ABB RAPID module: P105.mod

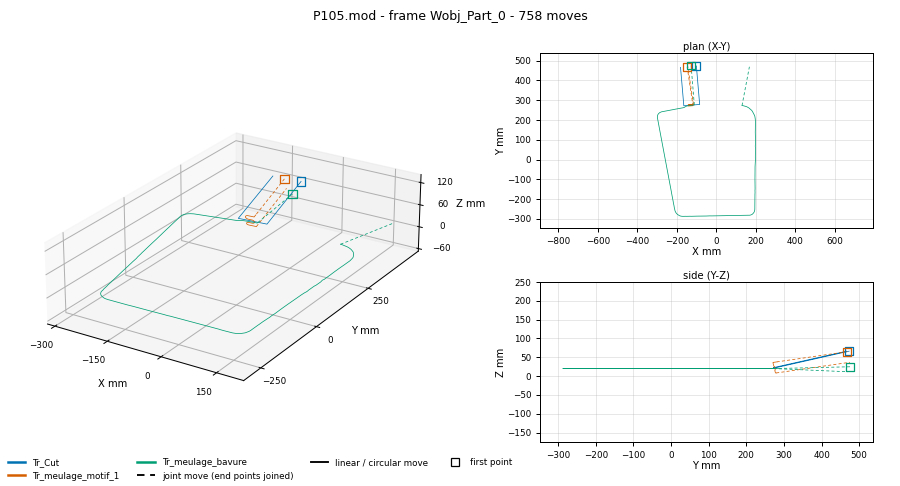
[picture p0: tool path of P105.mod in frame Wobj_Part_0, 758 of 766 moves have a stored position in this frame; points joined in program order, loops and branches not executed]
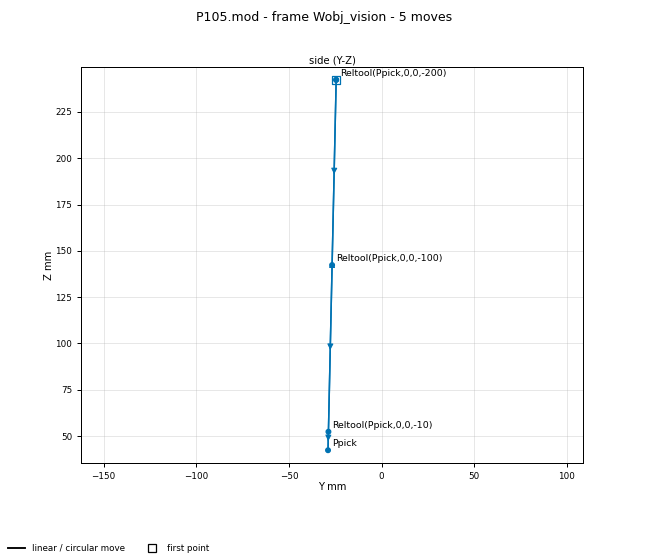
[picture p1: tool path of P105.mod in frame Wobj_vision, 5 of 766 moves have a stored position in this frame; points joined in program order, loops and branches not executed]
MODULE P105
	LOCAL CONST Speeddata vitesse_Tronconnage :=[10, 500, 0, 0];
	LOCAL CONST Robtarget Coupe_0 :=[[-129.483703125,274.966,22.39716015625],[0.465088414664095,0.570480739623642,-0.417793879465057,-0.532628169124803],[0,0,0,0],[8.999999E+09,8.999999E+09,8.999999E+09,8.999999E+09,8.999999E+09,8.999999E+09]];
	LOCAL CONST Robtarget Tr_meulage_motif_1_App1 :=[[-147.710429474566,468.187926503189,64.8611227493864],[0.0489177638432012,-0.0564309964361688,0.753506704297272,-0.653184691799237],[0,0,0,0],[8.999999E+09,8.999999E+09,8.999999E+09,8.999999E+09,8.999999E+09,8.999999E+09]];
	LOCAL CONST Robtarget Tr_meulage_motif_1_App2 :=[[-119.696933583103,282.208871325159,37.8975346530943],[0.0489177638432012,-0.0564309964361688,0.753506704297272,-0.653184691799237],[0,0,0,0],[8.999999E+09,8.999999E+09,8.999999E+09,8.999999E+09,8.999999E+09,8.999999E+09]];
	LOCAL CONST Robtarget Tr_meulage_motif_1_P0 :=[[-118.2225390625,272.4205,36.4783984375],[0.0489177638432012,-0.0564309964361688,0.753506704297272,-0.653184691799237],[0,0,0,0],[8.999999E+09,8.999999E+09,8.999999E+09,8.999999E+09,8.999999E+09,8.999999E+09]];
	LOCAL CONST Robtarget Tr_meulage_motif_1_P1 :=[[-119.2195859375,272.3438125,36.4796796875],[0.0489177638432012,-0.0564309964361688,0.753506704297272,-0.653184691799237],[0,0,0,0],[8.999999E+09,8.999999E+09,8.999999E+09,8.999999E+09,8.999999E+09,8.999999E+09]];
	LOCAL CONST Robtarget Tr_meulage_motif_1_P2 :=[[-120.216640625,272.267125,36.48095703125],[0.0489177638432012,-0.0564309964361688,0.753506704297272,-0.653184691799237],[0,0,0,0],[8.999999E+09,8.999999E+09,8.999999E+09,8.999999E+09,8.999999E+09,8.999999E+09]];
	LOCAL CONST Robtarget Tr_meulage_motif_1_P3 :=[[-121.2136953125,272.19040625,36.482234375],[0.0489177638432012,-0.0564309964361688,0.753506704297272,-0.653184691799237],[0,0,0,0],[8.999999E+09,8.999999E+09,8.999999E+09,8.999999E+09,8.999999E+09,8.999999E+09]];
	LOCAL CONST Robtarget Tr_meulage_motif_1_P4 :=[[-122.21075,272.11371875,36.483515625],[0.0489177638432012,-0.0564309964361688,0.753506704297272,-0.653184691799237],[0,0,0,0],[8.999999E+09,8.999999E+09,8.999999E+09,8.999999E+09,8.999999E+09,8.999999E+09]];
	LOCAL CONST Robtarget Tr_meulage_motif_1_P5 :=[[-123.2078046875,272.03703125,36.48479296875],[0.0489177638432012,-0.0564309964361688,0.753506704297272,-0.653184691799237],[0,0,0,0],[8.999999E+09,8.999999E+09,8.999999E+09,8.999999E+09,8.999999E+09,8.999999E+09]];
	LOCAL CONST Robtarget Tr_meulage_motif_1_P6 :=[[-124.204859375,271.9603125,36.4860703125],[0.0489177638432012,-0.0564309964361688,0.753506704297272,-0.653184691799237],[0,0,0,0],[8.999999E+09,8.999999E+09,8.999999E+09,8.999999E+09,8.999999E+09,8.999999E+09]];
	LOCAL CONST Robtarget Tr_meulage_motif_1_P7 :=[[-125.2019140625,271.883625,36.48734765625],[0.0489177638432012,-0.0564309964361688,0.753506704297272,-0.653184691799237],[0,0,0,0],[8.999999E+09,8.999999E+09,8.999999E+09,8.999999E+09,8.999999E+09,8.999999E+09]];
	LOCAL CONST Robtarget Tr_meulage_motif_1_P8 :=[[-126.1989609375,271.8069375,36.48862890625],[0.0489177638432012,-0.0564309964361688,0.753506704297272,-0.653184691799237],[0,0,0,0],[8.999999E+09,8.999999E+09,8.999999E+09,8.999999E+09,8.999999E+09,8.999999E+09]];
	LOCAL CONST Robtarget Tr_meulage_motif_1_P9 :=[[-127.196015625,271.73021875,36.48990625],[0.0489177638432012,-0.0564309964361688,0.753506704297272,-0.653184691799237],[0,0,0,0],[8.999999E+09,8.999999E+09,8.999999E+09,8.999999E+09,8.999999E+09,8.999999E+09]];
	LOCAL CONST Robtarget Tr_meulage_motif_1_P10 :=[[-128.1930703125,271.65353125,36.49118359375],[0.0489177638432012,-0.0564309964361688,0.753506704297272,-0.653184691799237],[0,0,0,0],[8.999999E+09,8.999999E+09,8.999999E+09,8.999999E+09,8.999999E+09,8.999999E+09]];
	LOCAL CONST Robtarget Tr_meulage_motif_1_P11 :=[[-129.190125,271.57684375,36.49246484375],[0.0489177638432012,-0.0564309964361688,0.753506704297272,-0.653184691799237],[0,0,0,0],[8.999999E+09,8.999999E+09,8.999999E+09,8.999999E+09,8.999999E+09,8.999999E+09]];
	LOCAL CONST Robtarget Tr_meulage_motif_1_P12 :=[[-130.1871796875,271.500125,36.4937421875],[0.0489177638432012,-0.0564309964361688,0.753506704297272,-0.653184691799237],[0,0,0,0],[8.999999E+09,8.999999E+09,8.999999E+09,8.999999E+09,8.999999E+09,8.999999E+09]];
	LOCAL CONST Robtarget Tr_meulage_motif_1_P13 :=[[-131.184234375,271.4234375,36.49501953125],[0.0489177638432012,-0.0564309964361688,0.753506704297272,-0.653184691799237],[0,0,0,0],[8.999999E+09,8.999999E+09,8.999999E+09,8.999999E+09,8.999999E+09,8.999999E+09]];
	LOCAL CONST Robtarget Tr_meulage_motif_1_P14 :=[[-132.18128125,271.34675,36.49630078125],[0.0489177638432012,-0.0564309964361688,0.753506704297272,-0.653184691799237],[0,0,0,0],[8.999999E+09,8.999999E+09,8.999999E+09,8.999999E+09,8.999999E+09,8.999999E+09]];
	LOCAL CONST Robtarget Tr_meulage_motif_1_P15 :=[[-133.17834375,271.27003125,36.497578125],[0.0489177638432012,-0.0564309964361688,0.753506704297272,-0.653184691799237],[0,0,0,0],[8.999999E+09,8.999999E+09,8.999999E+09,8.999999E+09,8.999999E+09,8.999999E+09]];
	LOCAL CONST Robtarget Tr_meulage_motif_1_P16 :=[[-134.175390625,271.19334375,36.49885546875],[0.0489177638432012,-0.0564309964361688,0.753506704297272,-0.653184691799237],[0,0,0,0],[8.999999E+09,8.999999E+09,8.999999E+09,8.999999E+09,8.999999E+09,8.999999E+09]];
	LOCAL CONST Robtarget Tr_meulage_motif_1_P17 :=[[-135.172453125,271.11665625,36.50013671875],[0.0489177638432012,-0.0564309964361688,0.753506704297272,-0.653184691799237],[0,0,0,0],[8.999999E+09,8.999999E+09,8.999999E+09,8.999999E+09,8.999999E+09,8.999999E+09]];
	LOCAL CONST Robtarget Tr_meulage_motif_1_P18 :=[[-136.1695,271.0399375,36.5014140625],[0.0489177638432012,-0.0564309964361688,0.753506704297272,-0.653184691799237],[0,0,0,0],[8.999999E+09,8.999999E+09,8.999999E+09,8.999999E+09,8.999999E+09,8.999999E+09]];
	LOCAL CONST Robtarget Tr_meulage_motif_1_P19 :=[[-137.161265625,270.9896875,36.39517578125],[0.0489177638432012,-0.0564309964361688,0.753506704297272,-0.653184691799237],[0,0,0,0],[8.999999E+09,8.999999E+09,8.999999E+09,8.999999E+09,8.999999E+09,8.999999E+09]];
	LOCAL CONST Robtarget Tr_meulage_motif_1_P20 :=[[-138.10903125,270.96646875,36.19109375],[0.0489177638432012,-0.0564309964361688,0.753506704297272,-0.653184691799237],[0,0,0,0],[8.999999E+09,8.999999E+09,8.999999E+09,8.999999E+09,8.999999E+09,8.999999E+09]];
	LOCAL CONST Robtarget Tr_meulage_motif_1_P21 :=[[-138.96446875,270.964625,35.92792578125],[0.0489177638432012,-0.0564309964361688,0.753506704297272,-0.653184691799237],[0,0,0,0],[8.999999E+09,8.999999E+09,8.999999E+09,8.999999E+09,8.999999E+09,8.999999E+09]];
	LOCAL CONST Robtarget Tr_meulage_motif_1_P22 :=[[-139.7175,270.971625,35.6606484375],[0.0489177638432012,-0.0564309964361688,0.753506704297272,-0.653184691799237],[0,0,0,0],[8.999999E+09,8.999999E+09,8.999999E+09,8.999999E+09,8.999999E+09,8.999999E+09]];
	LOCAL CONST Robtarget Tr_meulage_motif_1_P23 :=[[-140.827171875,271.03125,35.063125],[0.0489177638432012,-0.0564309964361688,0.753506704297272,-0.653184691799237],[0,0,0,0],[8.999999E+09,8.999999E+09,8.999999E+09,8.999999E+09,8.999999E+09,8.999999E+09]];
	LOCAL CONST Robtarget Tr_meulage_motif_1_P24 :=[[-141.86434375,271.15090625,34.2404375],[0.0489177638432012,-0.0564309964361688,0.753506704297272,-0.653184691799237],[0,0,0,0],[8.999999E+09,8.999999E+09,8.999999E+09,8.999999E+09,8.999999E+09,8.999999E+09]];
	LOCAL CONST Robtarget Tr_meulage_motif_1_P25 :=[[-142.7291875,271.32528125,33.24622265625],[0.0489177638432012,-0.0564309964361688,0.753506704297272,-0.653184691799237],[0,0,0,0],[8.999999E+09,8.999999E+09,8.999999E+09,8.999999E+09,8.999999E+09,8.999999E+09]];
	LOCAL CONST Robtarget Tr_meulage_motif_1_P26 :=[[-143.237375,271.5488125,32.16180859375],[0.0489177638432012,-0.0564309964361688,0.753506704297272,-0.653184691799237],[0,0,0,0],[8.999999E+09,8.999999E+09,8.999999E+09,8.999999E+09,8.999999E+09,8.999999E+09]];
	LOCAL CONST Robtarget Tr_meulage_motif_1_P27 :=[[-143.277734375,271.70946875,31.485298828125],[0.0489177638432012,-0.0564309964361688,0.753506704297272,-0.653184691799237],[0,0,0,0],[8.999999E+09,8.999999E+09,8.999999E+09,8.999999E+09,8.999999E+09,8.999999E+09]];
	LOCAL CONST Robtarget Tr_meulage_motif_1_P28 :=[[-143.290453125,271.86409375,30.84250390625],[0.0489177638432012,-0.0564309964361688,0.753506704297272,-0.653184691799237],[0,0,0,0],[8.999999E+09,8.999999E+09,8.999999E+09,8.999999E+09,8.999999E+09,8.999999E+09]];
	LOCAL CONST Robtarget Tr_meulage_motif_1_P29 :=[[-143.248453125,272.022875,30.1997890625],[0.0489177638432012,-0.0564309964361688,0.753506704297272,-0.653184691799237],[0,0,0,0],[8.999999E+09,8.999999E+09,8.999999E+09,8.999999E+09,8.999999E+09,8.999999E+09]];
	LOCAL CONST Robtarget Tr_meulage_motif_1_P30 :=[[-142.772890625,272.3186875,29.128150390625],[0.0489177638432012,-0.0564309964361688,0.753506704297272,-0.653184691799237],[0,0,0,0],[8.999999E+09,8.999999E+09,8.999999E+09,8.999999E+09,8.999999E+09,8.999999E+09]];
	LOCAL CONST Robtarget Tr_meulage_motif_1_P31 :=[[-141.93815625,272.61975,28.1485234375],[0.0489177638432012,-0.0564309964361688,0.753506704297272,-0.653184691799237],[0,0,0,0],[8.999999E+09,8.999999E+09,8.999999E+09,8.999999E+09,8.999999E+09,8.999999E+09]];
	LOCAL CONST Robtarget Tr_meulage_motif_1_P32 :=[[-140.933703125,272.89203125,27.34147265625],[0.0489177638432012,-0.0564309964361688,0.753506704297272,-0.653184691799237],[0,0,0,0],[8.999999E+09,8.999999E+09,8.999999E+09,8.999999E+09,8.999999E+09,8.999999E+09]];
	LOCAL CONST Robtarget Tr_meulage_motif_1_P33 :=[[-140.25625,273.03728125,26.955890625],[0.0489177638432012,-0.0564309964361688,0.753506704297272,-0.653184691799237],[0,0,0,0],[8.999999E+09,8.999999E+09,8.999999E+09,8.999999E+09,8.999999E+09,8.999999E+09]];
	LOCAL CONST Robtarget Tr_meulage_motif_1_P34 :=[[-139.110875,273.24009375,26.480484375],[0.0489177638432012,-0.0564309964361688,0.753506704297272,-0.653184691799237],[0,0,0,0],[8.999999E+09,8.999999E+09,8.999999E+09,8.999999E+09,8.999999E+09,8.999999E+09]];
	LOCAL CONST Robtarget Tr_meulage_motif_1_P35 :=[[-138.273421875,273.36665625,26.2226796875],[0.0489177638432012,-0.0564309964361688,0.753506704297272,-0.653184691799237],[0,0,0,0],[8.999999E+09,8.999999E+09,8.999999E+09,8.999999E+09,8.999999E+09,8.999999E+09]];
	LOCAL CONST Robtarget Tr_meulage_motif_1_P36 :=[[-137.34809375,273.4859375,26.0227265625],[0.0489177638432012,-0.0564309964361688,0.753506704297272,-0.653184691799237],[0,0,0,0],[8.999999E+09,8.999999E+09,8.999999E+09,8.999999E+09,8.999999E+09,8.999999E+09]];
	LOCAL CONST Robtarget Tr_meulage_motif_1_P37 :=[[-136.371515625,273.586625,25.915908203125],[0.0489177638432012,-0.0564309964361688,0.753506704297272,-0.653184691799237],[0,0,0,0],[8.999999E+09,8.999999E+09,8.999999E+09,8.999999E+09,8.999999E+09,8.999999E+09]];
	LOCAL CONST Robtarget Tr_meulage_motif_1_P38 :=[[-135.384,273.68859375,25.8071328125],[0.0489177638432012,-0.0564309964361688,0.753506704297272,-0.653184691799237],[0,0,0,0],[8.999999E+09,8.999999E+09,8.999999E+09,8.999999E+09,8.999999E+09,8.999999E+09]];
	LOCAL CONST Robtarget Tr_meulage_motif_1_P39 :=[[-134.386953125,273.76528125,25.805853515625],[0.0489177638432012,-0.0564309964361688,0.753506704297272,-0.653184691799237],[0,0,0,0],[8.999999E+09,8.999999E+09,8.999999E+09,8.999999E+09,8.999999E+09,8.999999E+09]];
	LOCAL CONST Robtarget Tr_meulage_motif_1_P40 :=[[-133.389890625,273.842,25.80457421875],[0.0489177638432012,-0.0564309964361688,0.753506704297272,-0.653184691799237],[0,0,0,0],[8.999999E+09,8.999999E+09,8.999999E+09,8.999999E+09,8.999999E+09,8.999999E+09]];
	LOCAL CONST Robtarget Tr_meulage_motif_1_P41 :=[[-132.39284375,273.9186875,25.803296875],[0.0489177638432012,-0.0564309964361688,0.753506704297272,-0.653184691799237],[0,0,0,0],[8.999999E+09,8.999999E+09,8.999999E+09,8.999999E+09,8.999999E+09,8.999999E+09]];
	LOCAL CONST Robtarget Tr_meulage_motif_1_P42 :=[[-131.395796875,273.995375,25.802017578125],[0.0489177638432012,-0.0564309964361688,0.753506704297272,-0.653184691799237],[0,0,0,0],[8.999999E+09,8.999999E+09,8.999999E+09,8.999999E+09,8.999999E+09,8.999999E+09]];
	LOCAL CONST Robtarget Tr_meulage_motif_1_P43 :=[[-130.398734375,274.07209375,25.80073828125],[0.0489177638432012,-0.0564309964361688,0.753506704297272,-0.653184691799237],[0,0,0,0],[8.999999E+09,8.999999E+09,8.999999E+09,8.999999E+09,8.999999E+09,8.999999E+09]];
	LOCAL CONST Robtarget Tr_meulage_motif_1_P44 :=[[-129.4016796875,274.14878125,25.7994609375],[0.0489177638432012,-0.0564309964361688,0.753506704297272,-0.653184691799237],[0,0,0,0],[8.999999E+09,8.999999E+09,8.999999E+09,8.999999E+09,8.999999E+09,8.999999E+09]];
	LOCAL CONST Robtarget Tr_meulage_motif_1_P45 :=[[-128.4046328125,274.22546875,25.798181640625],[0.0489177638432012,-0.0564309964361688,0.753506704297272,-0.653184691799237],[0,0,0,0],[8.999999E+09,8.999999E+09,8.999999E+09,8.999999E+09,8.999999E+09,8.999999E+09]];
	LOCAL CONST Robtarget Tr_meulage_motif_1_P46 :=[[-127.407578125,274.3021875,25.796904296875],[0.0489177638432012,-0.0564309964361688,0.753506704297272,-0.653184691799237],[0,0,0,0],[8.999999E+09,8.999999E+09,8.999999E+09,8.999999E+09,8.999999E+09,8.999999E+09]];
	LOCAL CONST Robtarget Tr_meulage_motif_1_P47 :=[[-126.4105234375,274.378875,25.795625],[0.0489177638432012,-0.0564309964361688,0.753506704297272,-0.653184691799237],[0,0,0,0],[8.999999E+09,8.999999E+09,8.999999E+09,8.999999E+09,8.999999E+09,8.999999E+09]];
	LOCAL CONST Robtarget Tr_meulage_motif_1_P48 :=[[-125.41346875,274.4555625,25.794345703125],[0.0489177638432012,-0.0564309964361688,0.753506704297272,-0.653184691799237],[0,0,0,0],[8.999999E+09,8.999999E+09,8.999999E+09,8.999999E+09,8.999999E+09,8.999999E+09]];
	LOCAL CONST Robtarget Tr_meulage_motif_1_P49 :=[[-124.4259609375,274.5575625,25.6855703125],[0.0489177638432012,-0.0564309964361688,0.753506704297272,-0.653184691799237],[0,0,0,0],[8.999999E+09,8.999999E+09,8.999999E+09,8.999999E+09,8.999999E+09,8.999999E+09]];
	LOCAL CONST Robtarget Tr_meulage_motif_1_P50 :=[[-123.4863046875,274.67953125,25.47906640625],[0.0489177638432012,-0.0564309964361688,0.753506704297272,-0.653184691799237],[0,0,0,0],[8.999999E+09,8.999999E+09,8.999999E+09,8.999999E+09,8.999999E+09,8.999999E+09]];
	LOCAL CONST Robtarget Tr_meulage_motif_1_P51 :=[[-122.641328125,274.8085,25.21371875],[0.0489177638432012,-0.0564309964361688,0.753506704297272,-0.653184691799237],[0,0,0,0],[8.999999E+09,8.999999E+09,8.999999E+09,8.999999E+09,8.999999E+09,8.999999E+09]];
	LOCAL CONST Robtarget Tr_meulage_motif_1_P52 :=[[-121.9377734375,274.9341875,24.917140625],[0.0489177638432012,-0.0564309964361688,0.753506704297272,-0.653184691799237],[0,0,0,0],[8.999999E+09,8.999999E+09,8.999999E+09,8.999999E+09,8.999999E+09,8.999999E+09]];
	LOCAL CONST Robtarget Tr_meulage_motif_1_P53 :=[[-120.91909375,275.1684375,24.27177734375],[0.0489177638432012,-0.0564309964361688,0.753506704297272,-0.653184691799237],[0,0,0,0],[8.999999E+09,8.999999E+09,8.999999E+09,8.999999E+09,8.999999E+09,8.999999E+09]];
	LOCAL CONST Robtarget Tr_meulage_motif_1_P54 :=[[-120.0371640625,275.4485,23.393859375],[0.0489177638432012,-0.0564309964361688,0.753506704297272,-0.653184691799237],[0,0,0,0],[8.999999E+09,8.999999E+09,8.999999E+09,8.999999E+09,8.999999E+09,8.999999E+09]];
	LOCAL CONST Robtarget Tr_meulage_motif_1_P55 :=[[-119.523890625,275.73409375,22.376337890625],[0.0489177638432012,-0.0564309964361688,0.753506704297272,-0.653184691799237],[0,0,0,0],[8.999999E+09,8.999999E+09,8.999999E+09,8.999999E+09,8.999999E+09,8.999999E+09]];
	LOCAL CONST Robtarget Tr_meulage_motif_1_P56 :=[[-119.352984375,275.91034375,21.702228515625],[0.0489177638432012,-0.0564309964361688,0.753506704297272,-0.653184691799237],[0,0,0,0],[8.999999E+09,8.999999E+09,8.999999E+09,8.999999E+09,8.999999E+09,8.999999E+09]];
	LOCAL CONST Robtarget Tr_meulage_motif_1_P57 :=[[-119.304140625,276.09528125,20.95363671875],[0.0489177638432012,-0.0564309964361688,0.753506704297272,-0.653184691799237],[0,0,0,0],[8.999999E+09,8.999999E+09,8.999999E+09,8.999999E+09,8.999999E+09,8.999999E+09]];
	LOCAL CONST Robtarget Tr_meulage_motif_1_P58 :=[[-119.3856875,276.27015625,20.205333984375],[0.0489177638432012,-0.0564309964361688,0.753506704297272,-0.653184691799237],[0,0,0,0],[8.999999E+09,8.999999E+09,8.999999E+09,8.999999E+09,8.999999E+09,8.999999E+09]];
	LOCAL CONST Robtarget Tr_meulage_motif_1_P59 :=[[-119.825359375,276.49709375,19.12855078125],[0.0489177638432012,-0.0564309964361688,0.753506704297272,-0.653184691799237],[0,0,0,0],[8.999999E+09,8.999999E+09,8.999999E+09,8.999999E+09,8.999999E+09,8.999999E+09]];
	LOCAL CONST Robtarget Tr_meulage_motif_1_P60 :=[[-120.2497109375,276.60228125,18.55973828125],[0.0489177638432012,-0.0564309964361688,0.753506704297272,-0.653184691799237],[0,0,0,0],[8.999999E+09,8.999999E+09,8.999999E+09,8.999999E+09,8.999999E+09,8.999999E+09]];
	LOCAL CONST Robtarget Tr_meulage_motif_1_P61 :=[[-121.1512890625,276.74165625,17.698505859375],[0.0489177638432012,-0.0564309964361688,0.753506704297272,-0.653184691799237],[0,0,0,0],[8.999999E+09,8.999999E+09,8.999999E+09,8.999999E+09,8.999999E+09,8.999999E+09]];
	LOCAL CONST Robtarget Tr_meulage_motif_1_P62 :=[[-121.74321875,276.79359375,17.296505859375],[0.0489177638432012,-0.0564309964361688,0.753506704297272,-0.653184691799237],[0,0,0,0],[8.999999E+09,8.999999E+09,8.999999E+09,8.999999E+09,8.999999E+09,8.999999E+09]];
	LOCAL CONST Robtarget Tr_meulage_motif_1_P63 :=[[-122.8682890625,276.8350625,16.76902734375],[0.0489177638432012,-0.0564309964361688,0.753506704297272,-0.653184691799237],[0,0,0,0],[8.999999E+09,8.999999E+09,8.999999E+09,8.999999E+09,8.999999E+09,8.999999E+09]];
	LOCAL CONST Robtarget Tr_meulage_motif_1_P64 :=[[-123.697140625,276.84084375,16.482830078125],[0.0489177638432012,-0.0564309964361688,0.753506704297272,-0.653184691799237],[0,0,0,0],[8.999999E+09,8.999999E+09,8.999999E+09,8.999999E+09,8.999999E+09,8.999999E+09]];
	LOCAL CONST Robtarget Tr_meulage_motif_1_P65 :=[[-124.6303203125,276.8171875,16.2852587890625],[0.0489177638432012,-0.0564309964361688,0.753506704297272,-0.653184691799237],[0,0,0,0],[8.999999E+09,8.999999E+09,8.999999E+09,8.999999E+09,8.999999E+09,8.999999E+09]];
	LOCAL CONST Robtarget Tr_meulage_motif_1_P66 :=[[-125.6110859375,276.76728125,16.1809501953125],[0.0489177638432012,-0.0564309964361688,0.753506704297272,-0.653184691799237],[0,0,0,0],[8.999999E+09,8.999999E+09,8.999999E+09,8.999999E+09,8.999999E+09,8.999999E+09]];
	LOCAL CONST Robtarget Tr_meulage_motif_1_P67 :=[[-126.60284375,276.717,16.074712890625],[0.0489177638432012,-0.0564309964361688,0.753506704297272,-0.653184691799237],[0,0,0,0],[8.999999E+09,8.999999E+09,8.999999E+09,8.999999E+09,8.999999E+09,8.999999E+09]];
	LOCAL CONST Robtarget Tr_meulage_motif_1_P68 :=[[-127.5998984375,276.6403125,16.0759912109375],[0.0489177638432012,-0.0564309964361688,0.753506704297272,-0.653184691799237],[0,0,0,0],[8.999999E+09,8.999999E+09,8.999999E+09,8.999999E+09,8.999999E+09,8.999999E+09]];
	LOCAL CONST Robtarget Tr_meulage_motif_1_P69 :=[[-128.596953125,276.563625,16.07726953125],[0.0489177638432012,-0.0564309964361688,0.753506704297272,-0.653184691799237],[0,0,0,0],[8.999999E+09,8.999999E+09,8.999999E+09,8.999999E+09,8.999999E+09,8.999999E+09]];
	LOCAL CONST Robtarget Tr_meulage_motif_1_P70 :=[[-129.5940078125,276.48690625,16.078548828125],[0.0489177638432012,-0.0564309964361688,0.753506704297272,-0.653184691799237],[0,0,0,0],[8.999999E+09,8.999999E+09,8.999999E+09,8.999999E+09,8.999999E+09,8.999999E+09]];
	LOCAL CONST Robtarget Tr_meulage_motif_1_P71 :=[[-130.5910625,276.41021875,16.0798271484375],[0.0489177638432012,-0.0564309964361688,0.753506704297272,-0.653184691799237],[0,0,0,0],[8.999999E+09,8.999999E+09,8.999999E+09,8.999999E+09,8.999999E+09,8.999999E+09]];
	LOCAL CONST Robtarget Tr_meulage_motif_1_P72 :=[[-131.588109375,276.33353125,16.08110546875],[0.0489177638432012,-0.0564309964361688,0.753506704297272,-0.653184691799237],[0,0,0,0],[8.999999E+09,8.999999E+09,8.999999E+09,8.999999E+09,8.999999E+09,8.999999E+09]];
	LOCAL CONST Robtarget Tr_meulage_motif_1_P73 :=[[-132.585171875,276.2568125,16.0823837890625],[0.0489177638432012,-0.0564309964361688,0.753506704297272,-0.653184691799237],[0,0,0,0],[8.999999E+09,8.999999E+09,8.999999E+09,8.999999E+09,8.999999E+09,8.999999E+09]];
	LOCAL CONST Robtarget Tr_meulage_motif_1_P74 :=[[-133.58221875,276.180125,16.0836630859375],[0.0489177638432012,-0.0564309964361688,0.753506704297272,-0.653184691799237],[0,0,0,0],[8.999999E+09,8.999999E+09,8.999999E+09,8.999999E+09,8.999999E+09,8.999999E+09]];
	LOCAL CONST Robtarget Tr_meulage_motif_1_P75 :=[[-134.57928125,276.1034375,16.08494140625],[0.0489177638432012,-0.0564309964361688,0.753506704297272,-0.653184691799237],[0,0,0,0],[8.999999E+09,8.999999E+09,8.999999E+09,8.999999E+09,8.999999E+09,8.999999E+09]];
	LOCAL CONST Robtarget Tr_meulage_motif_1_P76 :=[[-135.576328125,276.02671875,16.0862197265625],[0.0489177638432012,-0.0564309964361688,0.753506704297272,-0.653184691799237],[0,0,0,0],[8.999999E+09,8.999999E+09,8.999999E+09,8.999999E+09,8.999999E+09,8.999999E+09]];
	LOCAL CONST Robtarget Tr_meulage_motif_1_P77 :=[[-136.573390625,275.95003125,16.0874990234375],[0.0489177638432012,-0.0564309964361688,0.753506704297272,-0.653184691799237],[0,0,0,0],[8.999999E+09,8.999999E+09,8.999999E+09,8.999999E+09,8.999999E+09,8.999999E+09]];
	LOCAL CONST Robtarget Tr_meulage_motif_1_P78 :=[[-137.565140625,275.89978125,15.9812607421875],[0.0489177638432012,-0.0564309964361688,0.753506704297272,-0.653184691799237],[0,0,0,0],[8.999999E+09,8.999999E+09,8.999999E+09,8.999999E+09,8.999999E+09,8.999999E+09]];
	LOCAL CONST Robtarget Tr_meulage_motif_1_P79 :=[[-138.512921875,275.8765625,15.777177734375],[0.0489177638432012,-0.0564309964361688,0.753506704297272,-0.653184691799237],[0,0,0,0],[8.999999E+09,8.999999E+09,8.999999E+09,8.999999E+09,8.999999E+09,8.999999E+09]];
	LOCAL CONST Robtarget Tr_meulage_motif_1_P80 :=[[-139.368359375,275.87471875,15.5140107421875],[0.0489177638432012,-0.0564309964361688,0.753506704297272,-0.653184691799237],[0,0,0,0],[8.999999E+09,8.999999E+09,8.999999E+09,8.999999E+09,8.999999E+09,8.999999E+09]];
	LOCAL CONST Robtarget Tr_meulage_motif_1_P81 :=[[-140.121390625,275.88171875,15.2467333984375],[0.0489177638432012,-0.0564309964361688,0.753506704297272,-0.653184691799237],[0,0,0,0],[8.999999E+09,8.999999E+09,8.999999E+09,8.999999E+09,8.999999E+09,8.999999E+09]];
	LOCAL CONST Robtarget Tr_meulage_motif_1_P82 :=[[-141.2310625,275.9413125,14.6492109375],[0.0489177638432012,-0.0564309964361688,0.753506704297272,-0.653184691799237],[0,0,0,0],[8.999999E+09,8.999999E+09,8.999999E+09,8.999999E+09,8.999999E+09,8.999999E+09]];
	LOCAL CONST Robtarget Tr_meulage_motif_1_P83 :=[[-142.20215625,276.07696875,13.7814150390625],[0.0489177638432012,-0.0564309964361688,0.753506704297272,-0.653184691799237],[0,0,0,0],[8.999999E+09,8.999999E+09,8.999999E+09,8.999999E+09,8.999999E+09,8.999999E+09]];
	LOCAL CONST Robtarget Tr_meulage_motif_1_P84 :=[[-142.830375,276.28415625,12.7265029296875],[0.0489177638432012,-0.0564309964361688,0.753506704297272,-0.653184691799237],[0,0,0,0],[8.999999E+09,8.999999E+09,8.999999E+09,8.999999E+09,8.999999E+09,8.999999E+09]];
	LOCAL CONST Robtarget Tr_meulage_motif_1_P85 :=[[-143.018109375,276.50134375,11.7698173828125],[0.0489177638432012,-0.0564309964361688,0.753506704297272,-0.653184691799237],[0,0,0,0],[8.999999E+09,8.999999E+09,8.999999E+09,8.999999E+09,8.999999E+09,8.999999E+09]];
	LOCAL CONST Robtarget Tr_meulage_motif_1_P86 :=[[-142.89096875,276.55928125,11.570705078125],[0.0489177638432012,-0.0564309964361688,0.753506704297272,-0.653184691799237],[0,0,0,0],[8.999999E+09,8.999999E+09,8.999999E+09,8.999999E+09,8.999999E+09,8.999999E+09]];
	LOCAL CONST Robtarget Tr_meulage_motif_1_P87 :=[[-142.781921875,276.73859375,10.8644140625],[0.0489177638432012,-0.0564309964361688,0.753506704297272,-0.653184691799237],[0,0,0,0],[8.999999E+09,8.999999E+09,8.999999E+09,8.999999E+09,8.999999E+09,8.999999E+09]];
	LOCAL CONST Robtarget Tr_meulage_motif_1_P88 :=[[-142.11796875,277.01009375,9.95278125],[0.0489177638432012,-0.0564309964361688,0.753506704297272,-0.653184691799237],[0,0,0,0],[8.999999E+09,8.999999E+09,8.999999E+09,8.999999E+09,8.999999E+09,8.999999E+09]];
	LOCAL CONST Robtarget Tr_meulage_motif_1_P89 :=[[-141.57090625,277.1613125,9.5012001953125],[0.0489177638432012,-0.0564309964361688,0.753506704297272,-0.653184691799237],[0,0,0,0],[8.999999E+09,8.999999E+09,8.999999E+09,8.999999E+09,8.999999E+09,8.999999E+09]];
	LOCAL CONST Robtarget Tr_meulage_motif_1_P90 :=[[-140.454125,277.37203125,8.98412109375],[0.0489177638432012,-0.0564309964361688,0.753506704297272,-0.653184691799237],[0,0,0,0],[8.999999E+09,8.999999E+09,8.999999E+09,8.999999E+09,8.999999E+09,8.999999E+09]];
	LOCAL CONST Robtarget Tr_meulage_motif_1_P91 :=[[-139.61665625,277.49859375,8.7263173828125],[0.0489177638432012,-0.0564309964361688,0.753506704297272,-0.653184691799237],[0,0,0,0],[8.999999E+09,8.999999E+09,8.999999E+09,8.999999E+09,8.999999E+09,8.999999E+09]];
	LOCAL CONST Robtarget Tr_meulage_motif_1_P92 :=[[-138.69134375,277.617875,8.52636328125],[0.0489177638432012,-0.0564309964361688,0.753506704297272,-0.653184691799237],[0,0,0,0],[8.999999E+09,8.999999E+09,8.999999E+09,8.999999E+09,8.999999E+09,8.999999E+09]];
	LOCAL CONST Robtarget Tr_meulage_motif_1_P93 :=[[-137.71475,277.7185625,8.419544921875],[0.0489177638432012,-0.0564309964361688,0.753506704297272,-0.653184691799237],[0,0,0,0],[8.999999E+09,8.999999E+09,8.999999E+09,8.999999E+09,8.999999E+09,8.999999E+09]];
	LOCAL CONST Robtarget Tr_meulage_motif_1_P94 :=[[-136.72725,277.82053125,8.3107685546875],[0.0489177638432012,-0.0564309964361688,0.753506704297272,-0.653184691799237],[0,0,0,0],[8.999999E+09,8.999999E+09,8.999999E+09,8.999999E+09,8.999999E+09,8.999999E+09]];
	LOCAL CONST Robtarget Tr_meulage_motif_1_P95 :=[[-135.7301875,277.89725,8.309490234375],[0.0489177638432012,-0.0564309964361688,0.753506704297272,-0.653184691799237],[0,0,0,0],[8.999999E+09,8.999999E+09,8.999999E+09,8.999999E+09,8.999999E+09,8.999999E+09]];
	LOCAL CONST Robtarget Tr_meulage_motif_1_P96 :=[[-134.733140625,277.9739375,8.3082119140625],[0.0489177638432012,-0.0564309964361688,0.753506704297272,-0.653184691799237],[0,0,0,0],[8.999999E+09,8.999999E+09,8.999999E+09,8.999999E+09,8.999999E+09,8.999999E+09]];
	LOCAL CONST Robtarget Tr_meulage_motif_1_P97 :=[[-133.736078125,278.050625,8.3069326171875],[0.0489177638432012,-0.0564309964361688,0.753506704297272,-0.653184691799237],[0,0,0,0],[8.999999E+09,8.999999E+09,8.999999E+09,8.999999E+09,8.999999E+09,8.999999E+09]];
	LOCAL CONST Robtarget Tr_meulage_motif_1_P98 :=[[-132.73903125,278.12734375,8.305654296875],[0.0489177638432012,-0.0564309964361688,0.753506704297272,-0.653184691799237],[0,0,0,0],[8.999999E+09,8.999999E+09,8.999999E+09,8.999999E+09,8.999999E+09,8.999999E+09]];
	LOCAL CONST Robtarget Tr_meulage_motif_1_P99 :=[[-131.74196875,278.20403125,8.3043759765625],[0.0489177638432012,-0.0564309964361688,0.753506704297272,-0.653184691799237],[0,0,0,0],[8.999999E+09,8.999999E+09,8.999999E+09,8.999999E+09,8.999999E+09,8.999999E+09]];
	LOCAL CONST Robtarget Tr_meulage_motif_1_P100 :=[[-130.744921875,278.28071875,8.30309765625],[0.0489177638432012,-0.0564309964361688,0.753506704297272,-0.653184691799237],[0,0,0,0],[8.999999E+09,8.999999E+09,8.999999E+09,8.999999E+09,8.999999E+09,8.999999E+09]];
	LOCAL CONST Robtarget Tr_meulage_motif_1_P101 :=[[-129.7478671875,278.3574375,8.301818359375],[0.0489177638432012,-0.0564309964361688,0.753506704297272,-0.653184691799237],[0,0,0,0],[8.999999E+09,8.999999E+09,8.999999E+09,8.999999E+09,8.999999E+09,8.999999E+09]];
	LOCAL CONST Robtarget Tr_meulage_motif_1_P102 :=[[-128.7508125,278.434125,8.3005400390625],[0.0489177638432012,-0.0564309964361688,0.753506704297272,-0.653184691799237],[0,0,0,0],[8.999999E+09,8.999999E+09,8.999999E+09,8.999999E+09,8.999999E+09,8.999999E+09]];
	LOCAL CONST Robtarget Tr_meulage_motif_1_P103 :=[[-127.7537578125,278.5108125,8.29926171875],[0.0489177638432012,-0.0564309964361688,0.753506704297272,-0.653184691799237],[0,0,0,0],[8.999999E+09,8.999999E+09,8.999999E+09,8.999999E+09,8.999999E+09,8.999999E+09]];
	LOCAL CONST Robtarget Tr_meulage_motif_1_P104 :=[[-126.7567109375,278.58753125,8.297982421875],[0.0489177638432012,-0.0564309964361688,0.753506704297272,-0.653184691799237],[0,0,0,0],[8.999999E+09,8.999999E+09,8.999999E+09,8.999999E+09,8.999999E+09,8.999999E+09]];
	LOCAL CONST Robtarget Tr_meulage_motif_1_P105 :=[[-125.75965625,278.66421875,8.2967041015625],[0.0489177638432012,-0.0564309964361688,0.753506704297272,-0.653184691799237],[0,0,0,0],[8.999999E+09,8.999999E+09,8.999999E+09,8.999999E+09,8.999999E+09,8.999999E+09]];
	LOCAL CONST Robtarget Tr_meulage_motif_1_P106 :=[[-124.7626015625,278.74090625,8.29542578125],[0.0489177638432012,-0.0564309964361688,0.753506704297272,-0.653184691799237],[0,0,0,0],[8.999999E+09,8.999999E+09,8.999999E+09,8.999999E+09,8.999999E+09,8.999999E+09]];
	LOCAL CONST Robtarget Tr_meulage_motif_1_P107 :=[[-123.765546875,278.817625,8.294146484375],[0.0489177638432012,-0.0564309964361688,0.753506704297272,-0.653184691799237],[0,0,0,0],[8.999999E+09,8.999999E+09,8.999999E+09,8.999999E+09,8.999999E+09,8.999999E+09]];
	LOCAL CONST Robtarget Tr_meulage_motif_1_P108 :=[[-122.7684921875,278.8943125,8.2928681640625],[0.0489177638432012,-0.0564309964361688,0.753506704297272,-0.653184691799237],[0,0,0,0],[8.999999E+09,8.999999E+09,8.999999E+09,8.999999E+09,8.999999E+09,8.999999E+09]];
	LOCAL CONST Robtarget Tr_meulage_motif_1_P109 :=[[-121.7714375,278.971,8.29158984375],[0.0489177638432012,-0.0564309964361688,0.753506704297272,-0.653184691799237],[0,0,0,0],[8.999999E+09,8.999999E+09,8.999999E+09,8.999999E+09,8.999999E+09,8.999999E+09]];
	LOCAL CONST Robtarget Tr_meulage_motif_1_P110 :=[[-120.7743828125,279.04771875,8.2903115234375],[0.0489177638432012,-0.0564309964361688,0.753506704297272,-0.653184691799237],[0,0,0,0],[8.999999E+09,8.999999E+09,8.999999E+09,8.999999E+09,8.999999E+09,8.999999E+09]];
	LOCAL CONST Robtarget Tr_meulage_motif_1_P111 :=[[-119.7773359375,279.12440625,8.2890322265625],[0.0489177638432012,-0.0564309964361688,0.753506704297272,-0.653184691799237],[0,0,0,0],[8.999999E+09,8.999999E+09,8.999999E+09,8.999999E+09,8.999999E+09,8.999999E+09]];
	LOCAL CONST Robtarget Tr_meulage_motif_1_P112 :=[[-118.78028125,279.20109375,8.28775390625],[0.0489177638432012,-0.0564309964361688,0.753506704297272,-0.653184691799237],[0,0,0,0],[8.999999E+09,8.999999E+09,8.999999E+09,8.999999E+09,8.999999E+09,8.999999E+09]];
	LOCAL CONST Robtarget Tr_meulage_motif_1_P113 :=[[-117.7832265625,279.2778125,8.2864755859375],[0.0489177638432012,-0.0564309964361688,0.753506704297272,-0.653184691799237],[0,0,0,0],[8.999999E+09,8.999999E+09,8.999999E+09,8.999999E+09,8.999999E+09,8.999999E+09]];
	LOCAL CONST Robtarget Tr_meulage_motif_1_P114 :=[[-116.786171875,279.3545,8.2851962890625],[0.0489177638432012,-0.0564309964361688,0.753506704297272,-0.653184691799237],[0,0,0,0],[8.999999E+09,8.999999E+09,8.999999E+09,8.999999E+09,8.999999E+09,8.999999E+09]];
	LOCAL CONST Robtarget Tr_meulage_motif_1_P115 :=[[-115.7891171875,279.4311875,8.28391796875],[0.0489177638432012,-0.0564309964361688,0.753506704297272,-0.653184691799237],[0,0,0,0],[8.999999E+09,8.999999E+09,8.999999E+09,8.999999E+09,8.999999E+09,8.999999E+09]];
	LOCAL CONST Robtarget Tr_meulage_motif_1_degg1 :=[[-117.263511708103,289.219558825159,9.70305418434432],[0.0489177638432012,-0.0564309964361688,0.753506704297272,-0.653184691799237],[0,0,0,0],[8.999999E+09,8.999999E+09,8.999999E+09,8.999999E+09,8.999999E+09,8.999999E+09]];
	LOCAL CONST Robtarget Tr_meulage_motif_1_degg2 :=[[-145.277007599566,475.198614003189,36.6666422806364],[0.0489177638432012,-0.0564309964361688,0.753506704297272,-0.653184691799237],[0,0,0,0],[8.999999E+09,8.999999E+09,8.999999E+09,8.999999E+09,8.999999E+09,8.999999E+09]];
	LOCAL CONST Robtarget Tr_meulage_bavure_App1 :=[[-127.662761652857,475.675223369492,24.7637053380944],[0.0281615628538368,-0.0288405118824744,0.714896837466493,-0.698067090638424],[0,0,0,0],[8.999999E+09,8.999999E+09,8.999999E+09,8.999999E+09,8.999999E+09,8.999999E+09]];
	LOCAL CONST Robtarget Tr_meulage_bavure_App2 :=[[-112.361976363893,286.346393980975,20.2381852669047],[0.0281615628538368,-0.0288405118824744,0.714896837466493,-0.698067090638424],[0,0,0,0],[8.999999E+09,8.999999E+09,8.999999E+09,8.999999E+09,8.999999E+09,8.999999E+09]];
	LOCAL CONST Robtarget Tr_meulage_bavure_P0 :=[[-111.556671875,276.38171875,20],[0.0281615628538368,-0.0288405118824744,0.714896837466493,-0.698067090638424],[0,0,0,0],[8.999999E+09,8.999999E+09,8.999999E+09,8.999999E+09,8.999999E+09,8.999999E+09]];
	LOCAL CONST Robtarget Tr_meulage_bavure_P1 :=[[-113.4911796875,276.40778125,20],[0.0283477950994658,-0.0290312069301224,0.714888792871868,-0.698059886659721],[0,0,0,0],[8.999999E+09,8.999999E+09,8.999999E+09,8.999999E+09,8.999999E+09,8.999999E+09]];
	LOCAL CONST Robtarget Tr_meulage_bavure_P2 :=[[-114.227046875,276.36353125,20],[0.0289138852963095,-0.0296133534477701,0.714893347571618,-0.698007548764692],[0,0,0,0],[8.999999E+09,8.999999E+09,8.999999E+09,8.999999E+09,8.999999E+09,8.999999E+09]];
	LOCAL CONST Robtarget Tr_meulage_bavure_P3 :=[[-115.38265625,276.2895,20],[0.0298420341267732,-0.0305674601706369,0.714893262180734,-0.697927436820248],[0,0,0,0],[8.999999E+09,8.999999E+09,8.999999E+09,8.999999E+09,8.999999E+09,8.999999E+09]];
	LOCAL CONST Robtarget Tr_meulage_bavure_P4 :=[[-117.9585,275.97834375,20],[0.0311033066375073,-0.0318650497983372,0.714898654342968,-0.697808796832038],[0,0,0,0],[8.999999E+09,8.999999E+09,8.999999E+09,8.999999E+09,8.999999E+09,8.999999E+09]];
	LOCAL CONST Robtarget Tr_meulage_bavure_P5 :=[[-124.24475,275.153625,20],[0.0326905150815102,-0.0334987855508117,0.714903845284083,-0.697654394086612],[0,0,0,0],[8.999999E+09,8.999999E+09,8.999999E+09,8.999999E+09,8.999999E+09,8.999999E+09]];
	LOCAL CONST Robtarget Tr_meulage_bavure_P6 :=[[-125.3219921875,274.9531875,20],[0.0345928512087003,-0.0354581227392293,0.714907591487501,-0.697461964418564],[0,0,0,0],[8.999999E+09,8.999999E+09,8.999999E+09,8.999999E+09,8.999999E+09,8.999999E+09]];
	LOCAL CONST Robtarget Tr_meulage_bavure_P7 :=[[-125.4913671875,274.909,20],[0.0368179486486608,-0.0377512495688886,0.71490473966318,-0.697230589561597],[0,0,0,0],[8.999999E+09,8.999999E+09,8.999999E+09,8.999999E+09,8.999999E+09,8.999999E+09]];
	LOCAL CONST Robtarget Tr_meulage_bavure_P8 :=[[-125.6513046875,274.89496875,20],[0.03939764677674,-0.0404101260488098,0.714878629321826,-0.696967282216405],[0,0,0,0],[8.999999E+09,8.999999E+09,8.999999E+09,8.999999E+09,8.999999E+09,8.999999E+09]];
	LOCAL CONST Robtarget Tr_meulage_bavure_P9 :=[[-129.23946875,274.50859375,20],[0.0423999504940152,-0.0435067953611752,0.714835142168377,-0.696649210490202],[0,0,0,0],[8.999999E+09,8.999999E+09,8.999999E+09,8.999999E+09,8.999999E+09,8.999999E+09]];
	LOCAL CONST Robtarget Tr_meulage_bavure_P10 :=[[-132.406890625,274.05884375,20],[0.0459115778311491,-0.0471307554285718,0.714758640576694,-0.696269275952015],[0,0,0,0],[8.999999E+09,8.999999E+09,8.999999E+09,8.999999E+09,8.999999E+09,8.999999E+09]];
	LOCAL CONST Robtarget Tr_meulage_bavure_P11 :=[[-132.969140625,273.95428125,20],[0.0500378720218742,-0.0513915797670992,0.714634750910856,-0.695810527143089],[0,0,0,0],[8.999999E+09,8.999999E+09,8.999999E+09,8.999999E+09,8.999999E+09,8.999999E+09]];
	LOCAL CONST Robtarget Tr_meulage_bavure_P12 :=[[-134.00925,273.83671875,20],[0.0549072927302078,-0.0564229319432097,0.714442325196723,-0.69525089422702],[0,0,0,0],[8.999999E+09,8.999999E+09,8.999999E+09,8.999999E+09,8.999999E+09,8.999999E+09]];
	LOCAL CONST Robtarget Tr_meulage_bavure_P13 :=[[-138.2423125,273.13440625,20],[0.0606353943766575,-0.0623450147623814,0.714151230504875,-0.694567828258291],[0,0,0,0],[8.999999E+09,8.999999E+09,8.999999E+09,8.999999E+09,8.999999E+09,8.999999E+09]];
	LOCAL CONST Robtarget Tr_meulage_bavure_P14 :=[[-140.604,272.71534375,20],[0.0672951225867589,-0.0692341414725,0.713726832454981,-0.693737708910492],[0,0,0,0],[8.999999E+09,8.999999E+09,8.999999E+09,8.999999E+09,8.999999E+09,8.999999E+09]];
	LOCAL CONST Robtarget Tr_meulage_bavure_P15 :=[[-142.852015625,272.20946875,20],[0.0748956622598095,-0.0771011496135565,0.71313564484049,-0.69273631676192],[0,0,0,0],[8.999999E+09,8.999999E+09,8.999999E+09,8.999999E+09,8.999999E+09,8.999999E+09]];
	LOCAL CONST Robtarget Tr_meulage_bavure_P16 :=[[-146.281515625,271.63415625,20],[0.0833249016160749,-0.0858332119449677,0.71236058286735,-0.691543216635642],[0,0,0,0],[8.999999E+09,8.999999E+09,8.999999E+09,8.999999E+09,8.999999E+09,8.999999E+09]];
	LOCAL CONST Robtarget Tr_meulage_bavure_P17 :=[[-146.5704375,271.56334375,20],[0.0922968620410979,-0.0951394673540817,0.711414580991612,-0.69015872446958],[0,0,0,0],[8.999999E+09,8.999999E+09,8.999999E+09,8.999999E+09,8.999999E+09,8.999999E+09]];
	LOCAL CONST Robtarget Tr_meulage_bavure_P18 :=[[-149.573078125,270.7235,20],[0.10140080329549,-0.104596604725343,0.710330635498276,-0.688627486848714],[0,0,0,0],[8.999999E+09,8.999999E+09,8.999999E+09,8.999999E+09,8.999999E+09,8.999999E+09]];
	LOCAL CONST Robtarget Tr_meulage_bavure_P19 :=[[-150.456640625,270.50871875,20],[0.110071326993623,-0.113621698456806,0.709195132440937,-0.687034698349171],[0,0,0,0],[8.999999E+09,8.999999E+09,8.999999E+09,8.999999E+09,8.999999E+09,8.999999E+09]];
	LOCAL CONST Robtarget Tr_meulage_bavure_P20 :=[[-152.67553125,269.64921875,20],[0.117650351657146,-0.121538725290597,0.708152898886173,-0.68549704945302],[0,0,0,0],[8.999999E+09,8.999999E+09,8.999999E+09,8.999999E+09,8.999999E+09,8.999999E+09]];
	LOCAL CONST Robtarget Tr_meulage_bavure_P21 :=[[-153.696515625,269.0286875,20],[0.123517240347203,-0.127697017683855,0.707338082904325,-0.684185500785346],[0,0,0,0],[8.999999E+09,8.999999E+09,8.999999E+09,8.999999E+09,8.999999E+09,8.999999E+09]];
	LOCAL CONST Robtarget Tr_meulage_bavure_P22 :=[[-155.314921875,268.0153125,20],[0.127154287070356,-0.131557761294385,0.706900544780421,-0.683239315695447],[0,0,0,0],[8.999999E+09,8.999999E+09,8.999999E+09,8.999999E+09,8.999999E+09,8.999999E+09]];
	LOCAL CONST Robtarget Tr_meulage_bavure_P23 :=[[-158.761734375,265.4576875,20],[0.128232474048395,-0.132777023129003,0.706948666592096,-0.682751988303283],[0,0,0,0],[8.999999E+09,8.999999E+09,8.999999E+09,8.999999E+09,8.999999E+09,8.999999E+09]];
	LOCAL CONST Robtarget Tr_meulage_bavure_P24 :=[[-159.753390625,264.64990625,20],[0.126671523704774,-0.131264261920587,0.707509570788111,-0.682754879783351],[0,0,0,0],[8.999999E+09,8.999999E+09,8.999999E+09,8.999999E+09,8.999999E+09,8.999999E+09]];
	LOCAL CONST Robtarget Tr_meulage_bavure_P25 :=[[-160.19090625,264.44603125,20],[0.122679882853351,-0.127230560298217,0.708530579160486,-0.683188443450118],[0,0,0,0],[8.999999E+09,8.999999E+09,8.999999E+09,8.999999E+09,8.999999E+09,8.999999E+09]];
	LOCAL CONST Robtarget Tr_meulage_bavure_P26 :=[[-162.5858125,263.23546875,20],[0.116707170064269,-0.121133076952074,0.709879619484509,-0.683942351345668],[0,0,0,0],[8.999999E+09,8.999999E+09,8.999999E+09,8.999999E+09,8.999999E+09,8.999999E+09]];
	LOCAL CONST Robtarget Tr_meulage_bavure_P27 :=[[-164.2953125,262.84728125,20],[0.109374545489603,-0.113615640789659,0.711409734544896,-0.68485391475968],[0,0,0,0],[8.999999E+09,8.999999E+09,8.999999E+09,8.999999E+09,8.999999E+09,8.999999E+09]];
	LOCAL CONST Robtarget Tr_meulage_bavure_P28 :=[[-166.1201875,262.30378125,20],[0.101384105605423,-0.105399814464723,0.712953988312698,-0.685790604186444],[0,0,0,0],[8.999999E+09,8.999999E+09,8.999999E+09,8.999999E+09,8.999999E+09,8.999999E+09]];
	LOCAL CONST Robtarget Tr_meulage_bavure_P29 :=[[-169.657015625,261.750859375,20],[0.093430717692545,-0.0972071046556311,0.714389411111144,-0.686636183934548],[0,0,0,0],[8.999999E+09,8.999999E+09,8.999999E+09,8.999999E+09,8.999999E+09,8.999999E+09]];
	LOCAL CONST Robtarget Tr_meulage_bavure_P30 :=[[-169.824046875,261.719296875,20],[0.0860825966850136,-0.0896349363955776,0.715662988528616,-0.687300408537356],[0,0,0,0],[8.999999E+09,8.999999E+09,8.999999E+09,8.999999E+09,8.999999E+09,8.999999E+09]];
	LOCAL CONST Robtarget Tr_meulage_bavure_P31 :=[[-170.00609375,261.6926875,20],[0.0797263394006548,-0.0830835993299021,0.716735015108696,-0.687773032653431],[0,0,0,0],[8.999999E+09,8.999999E+09,8.999999E+09,8.999999E+09,8.999999E+09,8.999999E+09]];
	LOCAL CONST Robtarget Tr_meulage_bavure_P32 :=[[-173.3914375,261.00134375,20],[0.0745987625466033,-0.0778009746862547,0.717599932101635,-0.688064219686006],[0,0,0,0],[8.999999E+09,8.999999E+09,8.999999E+09,8.999999E+09,8.999999E+09,8.999999E+09]];
	LOCAL CONST Robtarget Tr_meulage_bavure_P33 :=[[-176.287265625,260.626890625,20],[0.0707485098392865,-0.0738429212613598,0.7182885884035,-0.688188473533535],[0,0,0,0],[8.999999E+09,8.999999E+09,8.999999E+09,8.999999E+09,8.999999E+09,8.999999E+09]];
	LOCAL CONST Robtarget Tr_meulage_bavure_P34 :=[[-180.45471875,259.89684375,20],[0.0680958490193906,-0.0711299194950713,0.718834222271648,-0.688172108407532],[0,0,0,0],[8.999999E+09,8.999999E+09,8.999999E+09,8.999999E+09,8.999999E+09,8.999999E+09]];
	LOCAL CONST Robtarget Tr_meulage_bavure_P35 :=[[-184.57084375,259.21490625,20],[0.0664898560341033,-0.0695060792475955,0.719261270575901,-0.688048856289822],[0,0,0,0],[8.999999E+09,8.999999E+09,8.999999E+09,8.999999E+09,8.999999E+09,8.999999E+09]];
	LOCAL CONST Robtarget Tr_meulage_bavure_P36 :=[[-185.099765625,259.09503125,20],[0.0657365700960871,-0.0687702739507533,0.719592560636171,-0.687848747509087],[0,0,0,0],[8.999999E+09,8.999999E+09,8.999999E+09,8.999999E+09,8.999999E+09,8.999999E+09]];
	LOCAL CONST Robtarget Tr_meulage_bavure_P37 :=[[-185.50546875,259.03375,20],[0.0656263240122323,-0.0687062514307359,0.719857648140777,-0.687588251080694],[0,0,0,0],[8.999999E+09,8.999999E+09,8.999999E+09,8.999999E+09,8.999999E+09,8.999999E+09]];
	LOCAL CONST Robtarget Tr_meulage_bavure_P38 :=[[-189.79215625,258.0885,20],[0.0659661167698859,-0.0691143083218761,0.720080976766236,-0.687280925621302],[0,0,0,0],[8.999999E+09,8.999999E+09,8.999999E+09,8.999999E+09,8.999999E+09,8.999999E+09]];
	LOCAL CONST Robtarget Tr_meulage_bavure_P39 :=[[-192.67665625,257.58215625,20],[0.0665898056937688,-0.0698161497902388,0.720253425404832,-0.686969072228684],[0,0,0,0],[8.999999E+09,8.999999E+09,8.999999E+09,8.999999E+09,8.999999E+09,8.999999E+09]];
	LOCAL CONST Robtarget Tr_meulage_bavure_P40 :=[[-194.422625,257.189265625,20],[0.0673336600015566,-0.0706464314399749,0.720419533219773,-0.686637426966369],[0,0,0,0],[8.999999E+09,8.999999E+09,8.999999E+09,8.999999E+09,8.999999E+09,8.999999E+09]];
	LOCAL CONST Robtarget Tr_meulage_bavure_P41 :=[[-196.795953125,256.828375,20],[0.0680779030394028,-0.0714777842800439,0.720582166672412,-0.686307268317818],[0,0,0,0],[8.999999E+09,8.999999E+09,8.999999E+09,8.999999E+09,8.999999E+09,8.999999E+09]];
	LOCAL CONST Robtarget Tr_meulage_bavure_P42 :=[[-199.052734375,256.358765625,20],[0.068733978004291,-0.0722154673844367,0.72074276680551,-0.685995940684558],[0,0,0,0],[8.999999E+09,8.999999E+09,8.999999E+09,8.999999E+09,8.999999E+09,8.999999E+09]];
	LOCAL CONST Robtarget Tr_meulage_bavure_P43 :=[[-200.2705625,256.177984375,20],[0.0692378458631994,-0.0727948627431868,0.720922226638025,-0.685695392866028],[0,0,0,0],[8.999999E+09,8.999999E+09,8.999999E+09,8.999999E+09,8.999999E+09,8.999999E+09]];
	LOCAL CONST Robtarget Tr_meulage_bavure_P44 :=[[-202.852671875,255.646546875,20],[0.0695609179763404,-0.0731835947508067,0.721114812162474,-0.685418753631325],[0,0,0,0],[8.999999E+09,8.999999E+09,8.999999E+09,8.999999E+09,8.999999E+09,8.999999E+09]];
	LOCAL CONST Robtarget Tr_meulage_bavure_P45 :=[[-206.395921875,254.9996875,20],[0.0697275098707865,-0.0734053535102146,0.721311314457666,-0.68517130418503],[0,0,0,0],[8.999999E+09,8.999999E+09,8.999999E+09,8.999999E+09,8.999999E+09,8.999999E+09]];
	LOCAL CONST Robtarget Tr_meulage_bavure_P46 :=[[-206.579484375,254.94640625,20],[0.0697857969761008,-0.0735105942581133,0.721506963599316,-0.684948053906225],[0,0,0,0],[8.999999E+09,8.999999E+09,8.999999E+09,8.999999E+09,8.999999E+09,8.999999E+09]];
	LOCAL CONST Robtarget Tr_meulage_bavure_P47 :=[[-206.751765625,254.92821875,20],[0.0697888529344498,-0.0735584368304128,0.721711747163744,-0.684726826101487],[0,0,0,0],[8.999999E+09,8.999999E+09,8.999999E+09,8.999999E+09,8.999999E+09,8.999999E+09]];
	LOCAL CONST Robtarget Tr_meulage_bavure_P48 :=[[-212.7269375,253.734984375,20],[0.0698109528016706,-0.0736263507060281,0.721914200990544,-0.684503818659049],[0,0,0,0],[8.999999E+09,8.999999E+09,8.999999E+09,8.999999E+09,8.999999E+09,8.999999E+09]];
	LOCAL CONST Robtarget Tr_meulage_bavure_P49 :=[[-215.185890625,253.30859375,20],[0.0699253316430651,-0.0737901236462662,0.722099408699673,-0.684279116737065],[0,0,0,0],[8.999999E+09,8.999999E+09,8.999999E+09,8.999999E+09,8.999999E+09,8.999999E+09]];
	LOCAL CONST Robtarget Tr_meulage_bavure_P50 :=[[-217.571796875,252.81659375,20],[0.070187000624867,-0.0741095225567156,0.722268277735663,-0.684039544607225],[0,0,0,0],[8.999999E+09,8.999999E+09,8.999999E+09,8.999999E+09,8.999999E+09,8.999999E+09]];
	LOCAL CONST Robtarget Tr_meulage_bavure_P51 :=[[-219.414578125,252.4294375,20],[0.0706161967342211,-0.0746063260134324,0.722418948131397,-0.68378221113034],[0,0,0,0],[8.999999E+09,8.999999E+09,8.999999E+09,8.999999E+09,8.999999E+09,8.999999E+09]];
	LOCAL CONST Robtarget Tr_meulage_bavure_P52 :=[[-219.592265625,252.3746875,20],[0.0712142143507482,-0.0752784780733785,0.722534158799455,-0.683524744088556],[0,0,0,0],[8.999999E+09,8.999999E+09,8.999999E+09,8.999999E+09,8.999999E+09,8.999999E+09]];
	LOCAL CONST Robtarget Tr_meulage_bavure_P53 :=[[-222.298515625,251.924375,20],[0.0719503851218481,-0.0760949782061291,0.722622347223387,-0.683263960461832],[0,0,0,0],[8.999999E+09,8.999999E+09,8.999999E+09,8.999999E+09,8.999999E+09,8.999999E+09]];
	LOCAL CONST Robtarget Tr_meulage_bavure_P54 :=[[-223.00653125,251.839234375,20],[0.07276252809863,-0.0769958132160336,0.722714685750316,-0.682979313195297],[0,0,0,0],[8.999999E+09,8.999999E+09,8.999999E+09,8.999999E+09,8.999999E+09,8.999999E+09]];
	LOCAL CONST Robtarget Tr_meulage_bavure_P55 :=[[-226.733125,251.095578125,20],[0.0735839005522163,-0.0779067192871709,0.72280187513122,-0.682695687679528],[0,0,0,0],[8.999999E+09,8.999999E+09,8.999999E+09,8.999999E+09,8.999999E+09,8.999999E+09]];
	LOCAL CONST Robtarget Tr_meulage_bavure_P56 :=[[-230.826953125,250.357421875,20],[0.0743327673679463,-0.0787393470696765,0.722885802747175,-0.68243012177441],[0,0,0,0],[8.999999E+09,8.999999E+09,8.999999E+09,8.999999E+09,8.999999E+09,8.999999E+09]];
	LOCAL CONST Robtarget Tr_meulage_bavure_P57 :=[[-231.306640625,250.255796875,20],[0.0749399820455924,-0.0794221627516598,0.722983018936734,-0.682181554634821],[0,0,0,0],[8.999999E+09,8.999999E+09,8.999999E+09,8.999999E+09,8.999999E+09,8.999999E+09]];
	LOCAL CONST Robtarget Tr_meulage_bavure_P58 :=[[-232.27103125,250.087953125,20],[0.0753420822238503,-0.0798863845473871,0.72309613930418,-0.681963129159863],[0,0,0,0],[8.999999E+09,8.999999E+09,8.999999E+09,8.999999E+09,8.999999E+09,8.999999E+09]];
	LOCAL CONST Robtarget Tr_meulage_bavure_P59 :=[[-236.269515625,249.218265625,20],[0.0754784635412745,-0.0800688847113417,0.723239034714655,-0.68177509041292],[0,0,0,0],[8.999999E+09,8.999999E+09,8.999999E+09,8.999999E+09,8.999999E+09,8.999999E+09]];
	LOCAL CONST Robtarget Tr_meulage_bavure_P60 :=[[-238.3276875,248.95459375,20],[0.0753029031774892,-0.0799174644686594,0.723405863569174,-0.681635260384673],[0,0,0,0],[8.999999E+09,8.999999E+09,8.999999E+09,8.999999E+09,8.999999E+09,8.999999E+09]];
	LOCAL CONST Robtarget Tr_meulage_bavure_P61 :=[[-241.622484375,248.2863125,20],[0.0747629573545809,-0.0793818944673386,0.723627353574113,-0.681522169997204],[0,0,0,0],[8.999999E+09,8.999999E+09,8.999999E+09,8.999999E+09,8.999999E+09,8.999999E+09]];
	LOCAL CONST Robtarget Tr_meulage_bavure_P62 :=[[-244.996203125,247.8045625,20],[0.0738339213907227,-0.0784299278182792,0.723882420640663,-0.681462793967435],[0,0,0,0],[8.999999E+09,8.999999E+09,8.999999E+09,8.999999E+09,8.999999E+09,8.999999E+09]];
	LOCAL CONST Robtarget Tr_meulage_bavure_P63 :=[[-245.692484375,247.64684375,20],[0.0725033952992989,-0.077049549880869,0.724177877525717,-0.681449210312534],[0,0,0,0],[8.999999E+09,8.999999E+09,8.999999E+09,8.999999E+09,8.999999E+09,8.999999E+09]];
	LOCAL CONST Robtarget Tr_meulage_bavure_P64 :=[[-246.061921875,247.61059375,20],[0.070769925553522,-0.0752383375952855,0.724509755523509,-0.681481052080183],[0,0,0,0],[8.999999E+09,8.999999E+09,8.999999E+09,8.999999E+09,8.999999E+09,8.999999E+09]];
	LOCAL CONST Robtarget Tr_meulage_bavure_P65 :=[[-250.131,246.775578125,20],[0.0686777314258527,-0.0730437174769128,0.724873932270543,-0.681546599183058],[0,0,0,0],[8.999999E+09,8.999999E+09,8.999999E+09,8.999999E+09,8.999999E+09,8.999999E+09]];
	LOCAL CONST Robtarget Tr_meulage_bavure_P66 :=[[-252.055953125,246.382390625,20],[0.0663333060132661,-0.0705775038467076,0.725250840812208,-0.681637679684232],[0,0,0,0],[8.999999E+09,8.999999E+09,8.999999E+09,8.999999E+09,8.999999E+09,8.999999E+09]];
	LOCAL CONST Robtarget Tr_meulage_bavure_P67 :=[[-252.8366875,246.199640625,20],[0.0638854426032939,-0.0679977738934828,0.725622234061603,-0.681738458944749],[0,0,0,0],[8.999999E+09,8.999999E+09,8.999999E+09,8.999999E+09,8.999999E+09,8.999999E+09]];
	LOCAL CONST Robtarget Tr_meulage_bavure_P68 :=[[-254.878875,245.8623125,20],[0.0615524416868129,-0.065540189038347,0.725982316427524,-0.681810425835316],[0,0,0,0],[8.999999E+09,8.999999E+09,8.999999E+09,8.999999E+09,8.999999E+09,8.999999E+09]];
	LOCAL CONST Robtarget Tr_meulage_bavure_P69 :=[[-257.003453125,245.451484375,20],[0.0596089057172335,-0.0634934596409505,0.726286904782653,-0.681852396698325],[0,0,0,0],[8.999999E+09,8.999999E+09,8.999999E+09,8.999999E+09,8.999999E+09,8.999999E+09]];
	LOCAL CONST Robtarget Tr_meulage_bavure_P70 :=[[-259.899296875,244.712828125,20],[0.0583541681448741,-0.0621792823263008,0.726523699112257,-0.681829775338206],[0,0,0,0],[8.999999E+09,8.999999E+09,8.999999E+09,8.999999E+09,8.999999E+09,8.999999E+09]];
	LOCAL CONST Robtarget Tr_meulage_bavure_P71 :=[[-260.77209375,244.660828125,20],[0.0581082804111509,-0.0619376272478277,0.726656951240024,-0.681730763053217],[0,0,0,0],[8.999999E+09,8.999999E+09,8.999999E+09,8.999999E+09,8.999999E+09,8.999999E+09]];
	LOCAL CONST Robtarget Tr_meulage_bavure_P72 :=[[-263.08940625,244.15509375,20],[0.0591493837147807,-0.063068367247824,0.726673949452027,-0.681519407388116],[0,0,0,0],[8.999999E+09,8.999999E+09,8.999999E+09,8.999999E+09,8.999999E+09,8.999999E+09]];
	LOCAL CONST Robtarget Tr_meulage_bavure_P73 :=[[-265.101625,243.75409375,20],[0.0617248762777957,-0.0658343619328377,0.726531985823662,-0.681180702906734],[0,0,0,0],[8.999999E+09,8.999999E+09,8.999999E+09,8.999999E+09,8.999999E+09,8.999999E+09]];
	LOCAL CONST Robtarget Tr_meulage_bavure_P74 :=[[-266.9828125,243.434203125,20],[0.0659876558698539,-0.0704025935501545,0.726208981697509,-0.680668508891134],[0,0,0,0],[8.999999E+09,8.999999E+09,8.999999E+09,8.999999E+09,8.999999E+09,8.999999E+09]];
	LOCAL CONST Robtarget Tr_meulage_bavure_P75 :=[[-268.42540625,243.133234375,20],[0.071998310258207,-0.0768383823869114,0.725658912541443,-0.679949445886455],[0,0,0,0],[8.999999E+09,8.999999E+09,8.999999E+09,8.999999E+09,8.999999E+09,8.999999E+09]];
	LOCAL CONST Robtarget Tr_meulage_bavure_P76 :=[[-269.75865625,242.943546875,20],[0.0797674469832447,-0.0851542972315429,0.724828948080916,-0.678976359005739],[0,0,0,0],[8.999999E+09,8.999999E+09,8.999999E+09,8.999999E+09,8.999999E+09,8.999999E+09]];
	LOCAL CONST Robtarget Tr_meulage_bavure_P77 :=[[-274.5713125,242.099796875,20],[0.0892043195507635,-0.0952547421282183,0.7236657916563,-0.677699745803429],[0,0,0,0],[8.999999E+09,8.999999E+09,8.999999E+09,8.999999E+09,8.999999E+09,8.999999E+09]];
	LOCAL CONST Robtarget Tr_meulage_bavure_P78 :=[[-277.44421875,241.45984375,20],[0.10015865038266,-0.106980271578654,0.722116426205693,-0.676070509082003],[0,0,0,0],[8.999999E+09,8.999999E+09,8.999999E+09,8.999999E+09,8.999999E+09,8.999999E+09]];
	LOCAL CONST Robtarget Tr_meulage_bavure_P79 :=[[-277.81271875,241.371640625,20],[0.112452890981654,-0.120142469175205,0.720131646684572,-0.674040463068591],[0,0,0,0],[8.999999E+09,8.999999E+09,8.999999E+09,8.999999E+09,8.999999E+09,8.999999E+09]];
	LOCAL CONST Robtarget Tr_meulage_bavure_P80 :=[[-277.9975625,241.30609375,20],[0.125892757567347,-0.13453617235357,0.717671686723767,-0.671564130962637],[0,0,0,0],[8.999999E+09,8.999999E+09,8.999999E+09,8.999999E+09,8.999999E+09,8.999999E+09]];
	LOCAL CONST Robtarget Tr_meulage_bavure_P81 :=[[-280.43378125,240.37140625,20],[0.140280380300671,-0.149947468822321,0.714693962969445,-0.668617761349119],[0,0,0,0],[8.999999E+09,8.999999E+09,8.999999E+09,8.999999E+09,8.999999E+09,8.999999E+09]];
	LOCAL CONST Robtarget Tr_meulage_bavure_P82 :=[[-283.30175,239.229609375,20],[0.155445353550186,-0.16619724546848,0.711174546393266,-0.66516613129404],[0,0,0,0],[8.999999E+09,8.999999E+09,8.999999E+09,8.999999E+09,8.999999E+09,8.999999E+09]];
	LOCAL CONST Robtarget Tr_meulage_bavure_P83 :=[[-285.7314375,237.846125,20],[0.171268349632142,-0.183157123897214,0.707078184576758,-0.661181564530969],[0,0,0,0],[8.999999E+09,8.999999E+09,8.999999E+09,8.999999E+09,8.999999E+09,8.999999E+09]];
	LOCAL CONST Robtarget Tr_meulage_bavure_P84 :=[[-285.8613125,237.772515625,20],[0.187659740176955,-0.200732493138758,0.702372418131711,-0.656630241736419],[0,0,0,0],[8.999999E+09,8.999999E+09,8.999999E+09,8.999999E+09,8.999999E+09,8.999999E+09]];
	LOCAL CONST Robtarget Tr_meulage_bavure_P85 :=[[-288.26815625,236.0806875,20],[0.204595598080059,-0.218898050764741,0.697006239973098,-0.651464953820406],[0,0,0,0],[8.999999E+09,8.999999E+09,8.999999E+09,8.999999E+09,8.999999E+09,8.999999E+09]];
	LOCAL CONST Robtarget Tr_meulage_bavure_P86 :=[[-288.35784375,236.01203125,20],[0.22209055955762,-0.237667252343187,0.690909288636581,-0.645627148898431],[0,0,0,0],[8.999999E+09,8.999999E+09,8.999999E+09,8.999999E+09,8.999999E+09,8.999999E+09]];
	LOCAL CONST Robtarget Tr_meulage_bavure_P87 :=[[-290.72696875,233.99084375,20],[0.240163469270989,-0.257065365296168,0.68401049289095,-0.639037206747737],[0,0,0,0],[8.999999E+09,8.999999E+09,8.999999E+09,8.999999E+09,8.999999E+09,8.999999E+09]];
	LOCAL CONST Robtarget Tr_meulage_bavure_P88 :=[[-291.10959375,233.586296875,20],[0.258796899557143,-0.277073408378721,0.676237321958266,-0.631630885517579],[0,0,0,0],[8.999999E+09,8.999999E+09,8.999999E+09,8.999999E+09,8.999999E+09,8.999999E+09]];
	LOCAL CONST Robtarget Tr_meulage_bavure_P89 :=[[-292.7609375,231.87084375,20],[0.277938615104208,-0.297637348767811,0.667530039539542,-0.623350448114671],[0,0,0,0],[8.999999E+09,8.999999E+09,8.999999E+09,8.999999E+09,8.999999E+09,8.999999E+09]];
	LOCAL CONST Robtarget Tr_meulage_bavure_P90 :=[[-293.4808125,230.820125,20],[0.297473808354015,-0.318639359667669,0.657861546287612,-0.614163233782363],[0,0,0,0],[8.999999E+09,8.999999E+09,8.999999E+09,8.999999E+09,8.999999E+09,8.999999E+09]];
	LOCAL CONST Robtarget Tr_meulage_bavure_P91 :=[[-294.65028125,229.219546875,20],[0.317188194425109,-0.339838526210616,0.647257941385675,-0.604118020533665],[0,0,0,0],[8.999999E+09,8.999999E+09,8.999999E+09,8.999999E+09,8.999999E+09,8.999999E+09]];
	LOCAL CONST Robtarget Tr_meulage_bavure_P92 :=[[-295.4455625,227.838140625,20],[0.336816844600856,-0.360964537579457,0.635821983823663,-0.593286963188736],[0,0,0,0],[8.999999E+09,8.999999E+09,8.999999E+09,8.999999E+09,8.999999E+09,8.999999E+09]];
	LOCAL CONST Robtarget Tr_meulage_bavure_P93 :=[[-295.96809375,226.7995,20],[0.35609913697017,-0.381729181437123,0.62368109223472,-0.581805922862041],[0,0,0,0],[8.999999E+09,8.999999E+09,8.999999E+09,8.999999E+09,8.999999E+09,8.999999E+09]];
	LOCAL CONST Robtarget Tr_meulage_bavure_P94 :=[[-296.27871875,226.103875,20],[0.374789773199657,-0.401866168758007,0.611002499497052,-0.569835198913744],[0,0,0,0],[8.999999E+09,8.999999E+09,8.999999E+09,8.999999E+09,8.999999E+09,8.999999E+09]];
	LOCAL CONST Robtarget Tr_meulage_bavure_P95 :=[[-297.24821875,223.3930625,20],[0.392681066066082,-0.421170857764024,0.597978574642742,-0.557528755484196],[0,0,0,0],[8.999999E+09,8.999999E+09,8.999999E+09,8.999999E+09,8.999999E+09,8.999999E+09]];
	LOCAL CONST Robtarget Tr_meulage_bavure_P96 :=[[-297.5436875,222.421625,20],[0.409651331058364,-0.439514412877423,0.584765931369407,-0.545033644231982],[0,0,0,0],[8.999999E+09,8.999999E+09,8.999999E+09,8.999999E+09,8.999999E+09,8.999999E+09]];
	LOCAL CONST Robtarget Tr_meulage_bavure_P97 :=[[-297.6419375,222.14171875,20],[0.425621956688545,-0.456801442793012,0.571508803379337,-0.532499839912423],[0,0,0,0],[8.999999E+09,8.999999E+09,8.999999E+09,8.999999E+09,8.999999E+09,8.999999E+09]];
	LOCAL CONST Robtarget Tr_meulage_bavure_P98 :=[[-297.7078125,221.673953125,20],[0.440513717434658,-0.472946000982756,0.558374664153569,-0.52008410794573],[0,0,0,0],[8.999999E+09,8.999999E+09,8.999999E+09,8.999999E+09,8.999999E+09,8.999999E+09]];
	LOCAL CONST Robtarget Tr_meulage_bavure_P99 :=[[-298.25590625,217.627078125,20],[0.454250683288702,-0.48787713280081,0.545547905574191,-0.507946555008912],[0,0,0,0],[8.999999E+09,8.999999E+09,8.999999E+09,8.999999E+09,8.999999E+09,8.999999E+09]];
	LOCAL CONST Robtarget Tr_meulage_bavure_P100 :=[[-298.19753125,216.55584375,20],[0.466770084342512,-0.501518649756865,0.533216148582464,-0.496271368507008],[0,0,0,0],[8.999999E+09,8.999999E+09,8.999999E+09,8.999999E+09,8.999999E+09,8.999999E+09]];
	LOCAL CONST Robtarget Tr_meulage_bavure_P101 :=[[-298.18875,214.716484375,20],[0.477983316325575,-0.513787153185668,0.521609723365784,-0.485260761885858],[0,0,0,0],[8.999999E+09,8.999999E+09,8.999999E+09,8.999999E+09,8.999999E+09,8.999999E+09]];
	LOCAL CONST Robtarget Tr_meulage_bavure_P102 :=[[-297.96234375,211.50246875,20],[0.487819541252689,-0.524596744951233,0.510956505291364,-0.475135559665894],[0,0,0,0],[8.999999E+09,8.999999E+09,8.999999E+09,8.999999E+09,8.999999E+09,8.999999E+09]];
	LOCAL CONST Robtarget Tr_meulage_bavure_P103 :=[[-297.69625,208.821234375,20],[0.496247106522207,-0.533930876288365,0.501446708052937,-0.466055605692227],[0,0,0,0],[8.999999E+09,8.999999E+09,8.999999E+09,8.999999E+09,8.999999E+09,8.999999E+09]];
	LOCAL CONST Robtarget Tr_meulage_bavure_P104 :=[[-296.69959375,203.081421875,20],[0.503278159950923,-0.541787539110278,0.493219078867676,-0.458161867053734],[0,0,0,0],[8.999999E+09,8.999999E+09,8.999999E+09,8.999999E+09,8.999999E+09,8.999999E+09]];
	LOCAL CONST Robtarget Tr_meulage_bavure_P105 :=[[-296.6438125,202.837828125,20],[0.50897512600457,-0.548229387116676,0.486336985419142,-0.451514337340164],[0,0,0,0],[8.999999E+09,8.999999E+09,8.999999E+09,8.999999E+09,8.999999E+09,8.999999E+09]];
	LOCAL CONST Robtarget Tr_meulage_bavure_P106 :=[[-296.6084375,202.69425,20],[0.51345096958881,-0.553374512238165,0.480777560566979,-0.446091569398872],[0,0,0,0],[8.999999E+09,8.999999E+09,8.999999E+09,8.999999E+09,8.999999E+09,8.999999E+09]];
	LOCAL CONST Robtarget Tr_meulage_bavure_P107 :=[[-295.7685625,198.935421875,20],[0.516848930042147,-0.557393936055109,0.476446406507313,-0.44178954864228],[0,0,0,0],[8.999999E+09,8.999999E+09,8.999999E+09,8.999999E+09,8.999999E+09,8.999999E+09]];
	LOCAL CONST Robtarget Tr_meulage_bavure_P108 :=[[-295.604,198.221890625,20],[0.519353493081534,-0.560472433256021,0.473175174650298,-0.438460779179557],[0,0,0,0],[8.999999E+09,8.999999E+09,8.999999E+09,8.999999E+09,8.999999E+09,8.999999E+09]];
	LOCAL CONST Robtarget Tr_meulage_bavure_P109 :=[[-294.99665625,195.513796875,20],[0.521136401253141,-0.562802963336558,0.470782376908804,-0.435928468146566],[0,0,0,0],[8.999999E+09,8.999999E+09,8.999999E+09,8.999999E+09,8.999999E+09,8.999999E+09]];
	LOCAL CONST Robtarget Tr_meulage_bavure_P110 :=[[-294.767,194.182984375,20],[0.522385329169383,-0.564578546028021,0.469052406601203,-0.433998240889408],[0,0,0,0],[8.999999E+09,8.999999E+09,8.999999E+09,8.999999E+09,8.999999E+09,8.999999E+09]];
	LOCAL CONST Robtarget Tr_meulage_bavure_P111 :=[[-293.499375,186.92965625,20],[0.523241584935745,-0.565959006869557,0.467813242316229,-0.432503660852403],[0,0,0,0],[8.999999E+09,8.999999E+09,8.999999E+09,8.999999E+09,8.999999E+09,8.999999E+09]];
	LOCAL CONST Robtarget Tr_meulage_bavure_P112 :=[[-293.0800625,184.2475625,20],[0.52382123288544,-0.567068473370629,0.466920920606642,-0.431311391441646],[0,0,0,0],[8.999999E+09,8.999999E+09,8.999999E+09,8.999999E+09,8.999999E+09,8.999999E+09]];
	LOCAL CONST Robtarget Tr_meulage_bavure_P113 :=[[-292.560125,181.33059375,20],[0.52421438091261,-0.56800584950956,0.466260654152657,-0.430313420841681],[0,0,0,0],[8.999999E+09,8.999999E+09,8.999999E+09,8.999999E+09,8.999999E+09,8.999999E+09]];
	LOCAL CONST Robtarget Tr_meulage_bavure_P114 :=[[-292.15590625,179.061609375,20],[0.524472782840716,-0.568817511848921,0.465769060888913,-0.429457937628329],[0,0,0,0],[8.999999E+09,8.999999E+09,8.999999E+09,8.999999E+09,8.999999E+09,8.999999E+09]];
	LOCAL CONST Robtarget Tr_meulage_bavure_P115 :=[[-291.6714375,176.7550625,20],[0.524607685506745,-0.56953069422415,0.465428380476033,-0.428716674846304],[0,0,0,0],[8.999999E+09,8.999999E+09,8.999999E+09,8.999999E+09,8.999999E+09,8.999999E+09]];
	LOCAL CONST Robtarget Tr_meulage_bavure_P116 :=[[-290.24296875,169.845734375,20],[0.524628403929957,-0.570140979605996,0.465231436003189,-0.428093461896153],[0,0,0,0],[8.999999E+09,8.999999E+09,8.999999E+09,8.999999E+09,8.999999E+09,8.999999E+09]];
	LOCAL CONST Robtarget Tr_meulage_bavure_P117 :=[[-290.17996875,169.582359375,20],[0.524530688916607,-0.570644362124585,0.465184592283625,-0.427593105021599],[0,0,0,0],[8.999999E+09,8.999999E+09,8.999999E+09,8.999999E+09,8.999999E+09,8.999999E+09]];
	LOCAL CONST Robtarget Tr_meulage_bavure_P118 :=[[-290.16503125,169.5405,20],[0.524298691795063,-0.571033540089019,0.465306826455035,-0.427224923348033],[0,0,0,0],[8.999999E+09,8.999999E+09,8.999999E+09,8.999999E+09,8.999999E+09,8.999999E+09]];
	LOCAL CONST Robtarget Tr_meulage_bavure_P119 :=[[-290.15925,169.51565625,20],[0.523940246822181,-0.571299629652048,0.465593317640849,-0.426996737092371],[0,0,0,0],[8.999999E+09,8.999999E+09,8.999999E+09,8.999999E+09,8.999999E+09,8.999999E+09]];
	LOCAL CONST Robtarget Tr_meulage_bavure_P120 :=[[-289.9225,168.07409375,20],[0.523456814887077,-0.571466998940906,0.466035722430683,-0.426883048958684],[0,0,0,0],[8.999999E+09,8.999999E+09,8.999999E+09,8.999999E+09,8.999999E+09,8.999999E+09]];
	LOCAL CONST Robtarget Tr_meulage_bavure_P121 :=[[-289.609125,166.30234375,20],[0.522877014273271,-0.571539857769972,0.466603777622486,-0.426875548179297],[0,0,0,0],[8.999999E+09,8.999999E+09,8.999999E+09,8.999999E+09,8.999999E+09,8.999999E+09]];
	LOCAL CONST Robtarget Tr_meulage_bavure_P122 :=[[-288.387375,158.944421875,20],[0.52221305677917,-0.571547884035851,0.467276268036477,-0.42694195028528],[0,0,0,0],[8.999999E+09,8.999999E+09,8.999999E+09,8.999999E+09,8.999999E+09,8.999999E+09]];
	LOCAL CONST Robtarget Tr_meulage_bavure_P123 :=[[-287.75415625,155.33821875,20],[0.521490109027818,-0.571512813358154,0.468021098662575,-0.427056695955325],[0,0,0,0],[8.999999E+09,8.999999E+09,8.999999E+09,8.999999E+09,8.999999E+09,8.999999E+09]];
	LOCAL CONST Robtarget Tr_meulage_bavure_P124 :=[[-287.1458125,152.270328125,20],[0.52073102439589,-0.571455450463059,0.468808827943827,-0.427195682573696],[0,0,0,0],[8.999999E+09,8.999999E+09,8.999999E+09,8.999999E+09,8.999999E+09,8.999999E+09]];
	LOCAL CONST Robtarget Tr_meulage_bavure_P125 :=[[-286.374625,148.220578125,20],[0.519950919612103,-0.571394009434237,0.469618691977623,-0.42733852075658],[0,0,0,0],[8.999999E+09,8.999999E+09,8.999999E+09,8.999999E+09,8.999999E+09,8.999999E+09]];
	LOCAL CONST Robtarget Tr_meulage_bavure_P126 :=[[-286.13178125,147.27609375,20],[0.519157938456091,-0.571337421542096,0.470439780366366,-0.427475143993773],[0,0,0,0],[8.999999E+09,8.999999E+09,8.999999E+09,8.999999E+09,8.999999E+09,8.999999E+09]];
	LOCAL CONST Robtarget Tr_meulage_bavure_P127 :=[[-285.9593125,146.7800625,20],[0.518355845674321,-0.571296258656759,0.471265174929763,-0.427594360344555],[0,0,0,0],[8.999999E+09,8.999999E+09,8.999999E+09,8.999999E+09,8.999999E+09,8.999999E+09]];
	LOCAL CONST Robtarget Tr_meulage_bavure_P128 :=[[-284.91409375,141.490453125,20],[0.517563155808256,-0.57125957567536,0.472079318567405,-0.427705499064417],[0,0,0,0],[8.999999E+09,8.999999E+09,8.999999E+09,8.999999E+09,8.999999E+09,8.999999E+09]];
	LOCAL CONST Robtarget Tr_meulage_bavure_P129 :=[[-284.79528125,140.984921875,20],[0.516773954890506,-0.571234158383532,0.472886242031522,-0.427802311751571],[0,0,0,0],[8.999999E+09,8.999999E+09,8.999999E+09,8.999999E+09,8.999999E+09,8.999999E+09]];
	LOCAL CONST Robtarget Tr_meulage_bavure_P130 :=[[-284.77725,140.854796875,20],[0.515990951080599,-0.571220352226025,0.473683120379159,-0.427884270654551],[0,0,0,0],[8.999999E+09,8.999999E+09,8.999999E+09,8.999999E+09,8.999999E+09,8.999999E+09]];
	LOCAL CONST Robtarget Tr_meulage_bavure_P131 :=[[-284.17146875,137.773984375,20],[0.515215113923963,-0.571222661723136,0.474467679820141,-0.427946816700797],[0,0,0,0],[8.999999E+09,8.999999E+09,8.999999E+09,8.999999E+09,8.999999E+09,8.999999E+09]];
	LOCAL CONST Robtarget Tr_meulage_bavure_P132 :=[[-284.1065,137.407140625,20],[0.514443850333118,-0.571245568843026,0.475241258180076,-0.427985714078242],[0,0,0,0],[8.999999E+09,8.999999E+09,8.999999E+09,8.999999E+09,8.999999E+09,8.999999E+09]];
	LOCAL CONST Robtarget Tr_meulage_bavure_P133 :=[[-283.221125,132.29659375,20],[0.513678714217012,-0.571283406249846,0.476003947276712,-0.428006647706459],[0,0,0,0],[8.999999E+09,8.999999E+09,8.999999E+09,8.999999E+09,8.999999E+09,8.999999E+09]];
	LOCAL CONST Robtarget Tr_meulage_bavure_P134 :=[[-282.86765625,130.371609375,20],[0.512921729301949,-0.571326854987322,0.476756424985745,-0.428018966419721],[0,0,0,0],[8.999999E+09,8.999999E+09,8.999999E+09,8.999999E+09,8.999999E+09,8.999999E+09]];
	LOCAL CONST Robtarget Tr_meulage_bavure_P135 :=[[-281.68296875,123.3819296875,20],[0.512170832917414,-0.571366659907107,0.477503480181983,-0.428032246763456],[0,0,0,0],[8.999999E+09,8.999999E+09,8.999999E+09,8.999999E+09,8.999999E+09,8.999999E+09]];
	LOCAL CONST Robtarget Tr_meulage_bavure_P136 :=[[-280.72675,118.237671875,20],[0.511420956293109,-0.571397960105693,0.478251653567647,-0.428051787183638],[0,0,0,0],[8.999999E+09,8.999999E+09,8.999999E+09,8.999999E+09,8.999999E+09,8.999999E+09]];
	LOCAL CONST Robtarget Tr_meulage_bavure_P137 :=[[-280.28384375,115.809875,20],[0.510671139733599,-0.571417420542106,0.47900288473058,-0.428081014486716],[0,0,0,0],[8.999999E+09,8.999999E+09,8.999999E+09,8.999999E+09,8.999999E+09,8.999999E+09]];
	LOCAL CONST Robtarget Tr_meulage_bavure_P138 :=[[-280.17421875,115.5210546875,20],[0.509924683571509,-0.571442020901038,0.479748902289637,-0.428102586519775],[0,0,0,0],[8.999999E+09,8.999999E+09,8.999999E+09,8.999999E+09,8.999999E+09,8.999999E+09]];
	LOCAL CONST Robtarget Tr_meulage_bavure_P139 :=[[-279.594375,112.3970625,20],[0.509209226101695,-0.571474519360475,0.48046104003471,-0.42811216612401],[0,0,0,0],[8.999999E+09,8.999999E+09,8.999999E+09,8.999999E+09,8.999999E+09,8.999999E+09]];
	LOCAL CONST Robtarget Tr_meulage_bavure_P140 :=[[-279.58290625,112.3583046875,20],[0.508535348880426,-0.571552860625622,0.481117627633286,-0.428071202991103],[0,0,0,0],[8.999999E+09,8.999999E+09,8.999999E+09,8.999999E+09,8.999999E+09,8.999999E+09]];
	LOCAL CONST Robtarget Tr_meulage_bavure_P141 :=[[-279.4444375,111.4702734375,20],[0.5079420117473,-0.571702226453236,0.481672085766325,-0.427952659489385],[0,0,0,0],[8.999999E+09,8.999999E+09,8.999999E+09,8.999999E+09,8.999999E+09,8.999999E+09]];
	LOCAL CONST Robtarget Tr_meulage_bavure_P142 :=[[-279.0223125,109.2665078125,20],[0.507452537068222,-0.571946654901231,0.482093856325681,-0.427731762046438],[0,0,0,0],[8.999999E+09,8.999999E+09,8.999999E+09,8.999999E+09,8.999999E+09,8.999999E+09]];
	LOCAL CONST Robtarget Tr_meulage_bavure_P143 :=[[-278.959875,108.9123828125,20],[0.507081408252769,-0.572304772357599,0.482362685202075,-0.427389673326053],[0,0,0,0],[8.999999E+09,8.999999E+09,8.999999E+09,8.999999E+09,8.999999E+09,8.999999E+09]];
	LOCAL CONST Robtarget Tr_meulage_bavure_P144 :=[[-278.82725,108.04684375,20],[0.50683771476717,-0.572764225122119,0.482472638578122,-0.426938902342381],[0,0,0,0],[8.999999E+09,8.999999E+09,8.999999E+09,8.999999E+09,8.999999E+09,8.999999E+09]];
	LOCAL CONST Robtarget Tr_meulage_bavure_P145 :=[[-277.78021875,101.6076953125,20],[0.50669238330336,-0.573313330171404,0.482455934309988,-0.426392923955373],[0,0,0,0],[8.999999E+09,8.999999E+09,8.999999E+09,8.999999E+09,8.999999E+09,8.999999E+09]];
	LOCAL CONST Robtarget Tr_meulage_bavure_P146 :=[[-277.24296875,98.1990078125,20],[0.506612219301428,-0.573908637476564,0.482358458291833,-0.425797196795142],[0,0,0,0],[8.999999E+09,8.999999E+09,8.999999E+09,8.999999E+09,8.999999E+09,8.999999E+09]];
	LOCAL CONST Robtarget Tr_meulage_bavure_P147 :=[[-276.68621875,94.9294453125,20],[0.506554277627344,-0.574497116526234,0.482239193841317,-0.42520722811796],[0,0,0,0],[8.999999E+09,8.999999E+09,8.999999E+09,8.999999E+09,8.999999E+09,8.999999E+09]];
	LOCAL CONST Robtarget Tr_meulage_bavure_P148 :=[[-276.22890625,92.9125703125,20],[0.506470026679006,-0.575033215886534,0.482160989918419,-0.424671275816776],[0,0,0,0],[8.999999E+09,8.999999E+09,8.999999E+09,8.999999E+09,8.999999E+09,8.999999E+09]];
	LOCAL CONST Robtarget Tr_meulage_bavure_P149 :=[[-275.42028125,88.775421875,20],[0.506336244489268,-0.575465645628117,0.482163352659049,-0.424242147329688],[0,0,0,0],[8.999999E+09,8.999999E+09,8.999999E+09,8.999999E+09,8.999999E+09,8.999999E+09]];
	LOCAL CONST Robtarget Tr_meulage_bavure_P150 :=[[-275.37984375,88.606625,20],[0.506132875133325,-0.575767823385483,0.482275240162492,-0.423947542733093],[0,0,0,0],[8.999999E+09,8.999999E+09,8.999999E+09,8.999999E+09,8.999999E+09,8.999999E+09]];
	LOCAL CONST Robtarget Tr_meulage_bavure_P151 :=[[-274.71328125,85.7136875,20],[0.50584543185462,-0.575946537435799,0.482509612358217,-0.423781145250057],[0,0,0,0],[8.999999E+09,8.999999E+09,8.999999E+09,8.999999E+09,8.999999E+09,8.999999E+09]];
	LOCAL CONST Robtarget Tr_meulage_bavure_P152 :=[[-274.22846875,83.6077890625,20],[0.505503195562424,-0.576007829273703,0.482835336019308,-0.423735221786785],[0,0,0,0],[8.999999E+09,8.999999E+09,8.999999E+09,8.999999E+09,8.999999E+09,8.999999E+09]];
	LOCAL CONST Robtarget Tr_meulage_bavure_P153 :=[[-273.682375,80.602234375,20],[0.505117933369315,-0.575988096525448,0.483229352412193,-0.423772319786222],[0,0,0,0],[8.999999E+09,8.999999E+09,8.999999E+09,8.999999E+09,8.999999E+09,8.999999E+09]];
	LOCAL CONST Robtarget Tr_meulage_bavure_P154 :=[[-272.9983125,76.5987578125,20],[0.504731972095412,-0.575912970464346,0.483641080242193,-0.423864591936829],[0,0,0,0],[8.999999E+09,8.999999E+09,8.999999E+09,8.999999E+09,8.999999E+09,8.999999E+09]];
	LOCAL CONST Robtarget Tr_meulage_bavure_P155 :=[[-272.611,74.313171875,20],[0.504367695939663,-0.575819469995633,0.484036523863428,-0.423973830363],[0,0,0,0],[8.999999E+09,8.999999E+09,8.999999E+09,8.999999E+09,8.999999E+09,8.999999E+09]];
	LOCAL CONST Robtarget Tr_meulage_bavure_P156 :=[[-272.35778125,73.051578125,20],[0.504055296218997,-0.575723817477316,0.484380308443008,-0.424082611215766],[0,0,0,0],[8.999999E+09,8.999999E+09,8.999999E+09,8.999999E+09,8.999999E+09,8.999999E+09]];
	LOCAL CONST Robtarget Tr_meulage_bavure_P157 :=[[-271.67471875,69.7786875,20],[0.503805366215231,-0.575646748971333,0.484655435454265,-0.424169874291078],[0,0,0,0],[8.999999E+09,8.999999E+09,8.999999E+09,8.999999E+09,8.999999E+09,8.999999E+09]];
	LOCAL CONST Robtarget Tr_meulage_bavure_P158 :=[[-270.9818125,66.6375703125,20],[0.503625829893903,-0.575600070766548,0.484850361334148,-0.424223654587258],[0,0,0,0],[8.999999E+09,8.999999E+09,8.999999E+09,8.999999E+09,8.999999E+09,8.999999E+09]];
	LOCAL CONST Robtarget Tr_meulage_bavure_P159 :=[[-270.76740625,65.8424375,20],[0.503519339834958,-0.575587842694767,0.484961217641611,-0.424239940526252],[0,0,0,0],[8.999999E+09,8.999999E+09,8.999999E+09,8.999999E+09,8.999999E+09,8.999999E+09]];
	LOCAL CONST Robtarget Tr_meulage_bavure_P160 :=[[-269.91153125,61.99462890625,20],[0.503489829851783,-0.575610910113241,0.484983810653359,-0.424217838850014],[0,0,0,0],[8.999999E+09,8.999999E+09,8.999999E+09,8.999999E+09,8.999999E+09,8.999999E+09]];
	LOCAL CONST Robtarget Tr_meulage_bavure_P161 :=[[-269.8015,61.7080390625,20],[0.503532325986964,-0.575678469567235,0.484920308841306,-0.424148311839309],[0,0,0,0],[8.999999E+09,8.999999E+09,8.999999E+09,8.999999E+09,8.999999E+09,8.999999E+09]];
	LOCAL CONST Robtarget Tr_meulage_bavure_P162 :=[[-269.2860625,58.59026953125,20],[0.503658041939778,-0.575782646865983,0.484761811147837,-0.424038803424947],[0,0,0,0],[8.999999E+09,8.999999E+09,8.999999E+09,8.999999E+09,8.999999E+09,8.999999E+09]];
	LOCAL CONST Robtarget Tr_meulage_bavure_P163 :=[[-269.26565625,58.5309453125,20],[0.503868838872078,-0.575921322978159,0.484507024676144,-0.423891219527206],[0,0,0,0],[8.999999E+09,8.999999E+09,8.999999E+09,8.999999E+09,8.999999E+09,8.999999E+09]];
	LOCAL CONST Robtarget Tr_meulage_bavure_P164 :=[[-269.10925,57.3551328125,20],[0.504156301143933,-0.576086047811402,0.484166926923692,-0.423714144686221],[0,0,0,0],[8.999999E+09,8.999999E+09,8.999999E+09,8.999999E+09,8.999999E+09,8.999999E+09]];
	LOCAL CONST Robtarget Tr_meulage_bavure_P165 :=[[-268.30884375,52.48641796875,20],[0.504495361841969,-0.576275096163812,0.483767174757835,-0.42351005188561],[0,0,0,0],[8.999999E+09,8.999999E+09,8.999999E+09,8.999999E+09,8.999999E+09,8.999999E+09]];
	LOCAL CONST Robtarget Tr_meulage_bavure_P166 :=[[-268.24025,51.971984375,20],[0.504874251177071,-0.57644453981398,0.483333178466019,-0.423323424358936],[0,0,0,0],[8.999999E+09,8.999999E+09,8.999999E+09,8.999999E+09,8.999999E+09,8.999999E+09]];
	LOCAL CONST Robtarget Tr_meulage_bavure_P167 :=[[-267.8826875,49.7984609375,20],[0.505261020738671,-0.576573633093645,0.482903586706221,-0.42317640823843],[0,0,0,0],[8.999999E+09,8.999999E+09,8.999999E+09,8.999999E+09,8.999999E+09,8.999999E+09]];
	LOCAL CONST Robtarget Tr_meulage_bavure_P168 :=[[-266.77978125,43.5256953125,20],[0.505625642815353,-0.576639693690196,0.482515787307583,-0.423093237936251],[0,0,0,0],[8.999999E+09,8.999999E+09,8.999999E+09,8.999999E+09,8.999999E+09,8.999999E+09]];
	LOCAL CONST Robtarget Tr_meulage_bavure_P169 :=[[-265.92946875,39.14990234375,20],[0.50594844217528,-0.576605320270876,0.482201348437297,-0.423112677736061],[0,0,0,0],[8.999999E+09,8.999999E+09,8.999999E+09,8.999999E+09,8.999999E+09,8.999999E+09]];
	LOCAL CONST Robtarget Tr_meulage_bavure_P170 :=[[-265.64590625,37.79803515625,20],[0.506224732981081,-0.576458168269311,0.48196883414111,-0.423247614134425],[0,0,0,0],[8.999999E+09,8.999999E+09,8.999999E+09,8.999999E+09,8.999999E+09,8.999999E+09]];
	LOCAL CONST Robtarget Tr_meulage_bavure_P171 :=[[-265.3798125,36.60198828125,20],[0.506454435969506,-0.576209542491982,0.481814646695478,-0.423486851812074],[0,0,0,0],[8.999999E+09,8.999999E+09,8.999999E+09,8.999999E+09,8.999999E+09,8.999999E+09]];
	LOCAL CONST Robtarget Tr_meulage_bavure_P172 :=[[-264.71971875,33.17590234375,20],[0.506655382438938,-0.575895150556639,0.481709496673294,-0.423793652413249],[0,0,0,0],[8.999999E+09,8.999999E+09,8.999999E+09,8.999999E+09,8.999999E+09,8.999999E+09]];
	LOCAL CONST Robtarget Tr_meulage_bavure_P173 :=[[-264.24175,30.47540234375,20],[0.506875577593424,-0.575552870061198,0.481593112063791,-0.424127477318275],[0,0,0,0],[8.999999E+09,8.999999E+09,8.999999E+09,8.999999E+09,8.999999E+09,8.999999E+09]];
	LOCAL CONST Robtarget Tr_meulage_bavure_P174 :=[[-263.0254375,24.30450390625,20],[0.507166619940553,-0.575242095449999,0.481395181228499,-0.424425765865304],[0,0,0,0],[8.999999E+09,8.999999E+09,8.999999E+09,8.999999E+09,8.999999E+09,8.999999E+09]];
	LOCAL CONST Robtarget Tr_meulage_bavure_P175 :=[[-262.75359375,22.749328125,20],[0.507572871054023,-0.575028084248357,0.481051149606142,-0.424620153028857],[0,0,0,0],[8.999999E+09,8.999999E+09,8.999999E+09,8.999999E+09,8.999999E+09,8.999999E+09]];
	LOCAL CONST Robtarget Tr_meulage_bavure_P176 :=[[-262.43365625,20.88397265625,20],[0.508136281585532,-0.574956661697104,0.480504891919847,-0.42466151856231],[0,0,0,0],[8.999999E+09,8.999999E+09,8.999999E+09,8.999999E+09,8.999999E+09,8.999999E+09]];
	LOCAL CONST Robtarget Tr_meulage_bavure_P177 :=[[-261.558875,16.3700869140625,20],[0.508885584058193,-0.575052200156239,0.47971988647826,-0.424522390399501],[0,0,0,0],[8.999999E+09,8.999999E+09,8.999999E+09,8.999999E+09,8.999999E+09,8.999999E+09]];
	LOCAL CONST Robtarget Tr_meulage_bavure_P178 :=[[-261.336296875,15.19790625,20],[0.509810990277013,-0.575310264718091,0.478706822413198,-0.424205883596432],[0,0,0,0],[8.999999E+09,8.999999E+09,8.999999E+09,8.999999E+09,8.999999E+09,8.999999E+09]];
	LOCAL CONST Robtarget Tr_meulage_bavure_P179 :=[[-261.01959375,13.762787109375,20],[0.510865306627209,-0.575701053532016,0.477521620080334,-0.42374289115296],[0,0,0,0],[8.999999E+09,8.999999E+09,8.999999E+09,8.999999E+09,8.999999E+09,8.999999E+09]];
	LOCAL CONST Robtarget Tr_meulage_bavure_P180 :=[[-259.358578125,4.8236083984375,20],[0.512016193707448,-0.57614391664705,0.476221033473116,-0.423215231259147],[0,0,0,0],[8.999999E+09,8.999999E+09,8.999999E+09,8.999999E+09,8.999999E+09,8.999999E+09]];
	LOCAL CONST Robtarget Tr_meulage_bavure_P181 :=[[-259.3125,4.670654296875,20],[0.51318932254815,-0.576577942824513,0.474898782149641,-0.422688705531165],[0,0,0,0],[8.999999E+09,8.999999E+09,8.999999E+09,8.999999E+09,8.999999E+09,8.999999E+09]];
	LOCAL CONST Robtarget Tr_meulage_bavure_P182 :=[[-259.15521875,3.76657104492188,20],[0.514312529864824,-0.576926777686543,0.473652009833001,-0.422246241420129],[0,0,0,0],[8.999999E+09,8.999999E+09,8.999999E+09,8.999999E+09,8.999999E+09,8.999999E+09]];
	LOCAL CONST Robtarget Tr_meulage_bavure_P183 :=[[-257.512390625,-4.14437890625,20],[0.515331046522538,-0.577128032332715,0.472556529863291,-0.421956719189681],[0,0,0,0],[8.999999E+09,8.999999E+09,8.999999E+09,8.999999E+09,8.999999E+09,8.999999E+09]];
	LOCAL CONST Robtarget Tr_meulage_bavure_P184 :=[[-256.93225,-7.30093359375,20],[0.516210124324792,-0.577156749717465,0.47165620538071,-0.421850231392639],[0,0,0,0],[8.999999E+09,8.999999E+09,8.999999E+09,8.999999E+09,8.999999E+09,8.999999E+09]];
	LOCAL CONST Robtarget Tr_meulage_bavure_P185 :=[[-256.265375,-10.523529296875,20],[0.516943377645753,-0.577007147283673,0.470959777459982,-0.421935047497364],[0,0,0,0],[8.999999E+09,8.999999E+09,8.999999E+09,8.999999E+09,8.999999E+09,8.999999E+09]];
	LOCAL CONST Robtarget Tr_meulage_bavure_P186 :=[[-255.981578125,-11.889892578125,20],[0.517546518358076,-0.576701215331517,0.470444338057924,-0.422188861008704],[0,0,0,0],[8.999999E+09,8.999999E+09,8.999999E+09,8.999999E+09,8.999999E+09,8.999999E+09]];
	LOCAL CONST Robtarget Tr_meulage_bavure_P187 :=[[-255.217625,-16.854552734375,20],[0.518065536784882,-0.576274183088468,0.470051758712492,-0.422572490388105],[0,0,0,0],[8.999999E+09,8.999999E+09,8.999999E+09,8.999999E+09,8.999999E+09,8.999999E+09]];
	LOCAL CONST Robtarget Tr_meulage_bavure_P188 :=[[-254.84421875,-19.565521484375,20],[0.518531498569311,-0.575777604160039,0.469733901218744,-0.42303108347379],[0,0,0,0],[8.999999E+09,8.999999E+09,8.999999E+09,8.999999E+09,8.999999E+09,8.999999E+09]];
	LOCAL CONST Robtarget Tr_meulage_bavure_P189 :=[[-254.42003125,-21.98175,20],[0.51898107907396,-0.575236591371339,0.469445376671715,-0.423535762164499],[0,0,0,0],[8.999999E+09,8.999999E+09,8.999999E+09,8.999999E+09,8.999999E+09,8.999999E+09]];
	LOCAL CONST Robtarget Tr_meulage_bavure_P190 :=[[-253.555171875,-26.341888671875,20],[0.519415793684495,-0.574685124418383,0.469173933413176,-0.424051955836714],[0,0,0,0],[8.999999E+09,8.999999E+09,8.999999E+09,8.999999E+09,8.999999E+09,8.999999E+09]];
	LOCAL CONST Robtarget Tr_meulage_bavure_P191 :=[[-252.96871875,-28.4684453125,20],[0.519842666457439,-0.574122199599636,0.468912681694941,-0.424580026618015],[0,0,0,0],[8.999999E+09,8.999999E+09,8.999999E+09,8.999999E+09,8.999999E+09,8.999999E+09]];
	LOCAL CONST Robtarget Tr_meulage_bavure_P192 :=[[-252.4610625,-31.030333984375,20],[0.520240781672039,-0.573543343150863,0.46868414402228,-0.425126729052291],[0,0,0,0],[8.999999E+09,8.999999E+09,8.999999E+09,8.999999E+09,8.999999E+09,8.999999E+09]];
	LOCAL CONST Robtarget Tr_meulage_bavure_P193 :=[[-252.028359375,-32.96875,20],[0.520604107048895,-0.572902941505298,0.468508027280063,-0.425739135753977],[0,0,0,0],[8.999999E+09,8.999999E+09,8.999999E+09,8.999999E+09,8.999999E+09,8.999999E+09]];
	LOCAL CONST Robtarget Tr_meulage_bavure_P194 :=[[-251.7274375,-34.70755078125,20],[0.520904753809199,-0.572189213580469,0.468415678459291,-0.426432284770588],[0,0,0,0],[8.999999E+09,8.999999E+09,8.999999E+09,8.999999E+09,8.999999E+09,8.999999E+09]];
	LOCAL CONST Robtarget Tr_meulage_bavure_P195 :=[[-251.448765625,-35.88848828125,20],[0.521123329505566,-0.571395133848023,0.46842820371117,-0.427215512859448],[0,0,0,0],[8.999999E+09,8.999999E+09,8.999999E+09,8.999999E+09,8.999999E+09,8.999999E+09]];
	LOCAL CONST Robtarget Tr_meulage_bavure_P196 :=[[-251.291359375,-36.5687578125,20],[0.521246824077857,-0.570512153365386,0.468560470944618,-0.428098956223086],[0,0,0,0],[8.999999E+09,8.999999E+09,8.999999E+09,8.999999E+09,8.999999E+09,8.999999E+09]];
	LOCAL CONST Robtarget Tr_meulage_bavure_P197 :=[[-250.47425,-41.8633125,20],[0.521286018124113,-0.56954664566529,0.468798675711047,-0.429074943770074],[0,0,0,0],[8.999999E+09,8.999999E+09,8.999999E+09,8.999999E+09,8.999999E+09,8.999999E+09]];
	LOCAL CONST Robtarget Tr_meulage_bavure_P198 :=[[-250.374609375,-42.3610234375,20],[0.521250845429041,-0.568520602567913,0.46912547615251,-0.430119946317312],[0,0,0,0],[8.999999E+09,8.999999E+09,8.999999E+09,8.999999E+09,8.999999E+09,8.999999E+09]];
	LOCAL CONST Robtarget Tr_meulage_bavure_P199 :=[[-249.878921875,-45.51240625,20],[0.521164947284982,-0.567454166685026,0.469510457885451,-0.431210849085965],[0,0,0,0],[8.999999E+09,8.999999E+09,8.999999E+09,8.999999E+09,8.999999E+09,8.999999E+09]];
	LOCAL CONST Robtarget Tr_meulage_bavure_P200 :=[[-249.30334375,-48.547484375,20],[0.521066812694018,-0.56637097997881,0.469907560459521,-0.432319528092038],[0,0,0,0],[8.999999E+09,8.999999E+09,8.999999E+09,8.999999E+09,8.999999E+09,8.999999E+09]];
	LOCAL CONST Robtarget Tr_meulage_bavure_P201 :=[[-249.153734375,-49.31654296875,20],[0.520971394175319,-0.565316286533165,0.470289273111373,-0.433398548945141],[0,0,0,0],[8.999999E+09,8.999999E+09,8.999999E+09,8.999999E+09,8.999999E+09,8.999999E+09]];
	LOCAL CONST Robtarget Tr_meulage_bavure_P202 :=[[-248.465953125,-52.32923828125,20],[0.520906356053275,-0.564320308509742,0.470619987095375,-0.434414531724156],[0,0,0,0],[8.999999E+09,8.999999E+09,8.999999E+09,8.999999E+09,8.999999E+09,8.999999E+09]];
	LOCAL CONST Robtarget Tr_meulage_bavure_P203 :=[[-247.831359375,-54.61175390625,20],[0.52089628021915,-0.563421666605151,0.47086553754631,-0.435326011633755],[0,0,0,0],[8.999999E+09,8.999999E+09,8.999999E+09,8.999999E+09,8.999999E+09,8.999999E+09]];
	LOCAL CONST Robtarget Tr_meulage_bavure_P204 :=[[-247.434140625,-56.24558984375,20],[0.520993131713762,-0.562657986033331,0.470964779342442,-0.436089811941218],[0,0,0,0],[8.999999E+09,8.999999E+09,8.999999E+09,8.999999E+09,8.999999E+09,8.999999E+09]];
	LOCAL CONST Robtarget Tr_meulage_bavure_P205 :=[[-246.824734375,-58.0758984375,20],[0.521237021282572,-0.562078667133239,0.470865859536226,-0.436651900169236],[0,0,0,0],[8.999999E+09,8.999999E+09,8.999999E+09,8.999999E+09,8.999999E+09,8.999999E+09]];
	LOCAL CONST Robtarget Tr_meulage_bavure_P206 :=[[-246.2899375,-60.47671484375,20],[0.521662184860214,-0.561722157457533,0.470525689727236,-0.436969516116205],[0,0,0,0],[8.999999E+09,8.999999E+09,8.999999E+09,8.999999E+09,8.999999E+09,8.999999E+09]];
	LOCAL CONST Robtarget Tr_meulage_bavure_P207 :=[[-246.066546875,-61.18641796875,20],[0.522303054886626,-0.561629028412525,0.469899975790022,-0.436996986320315],[0,0,0,0],[8.999999E+09,8.999999E+09,8.999999E+09,8.999999E+09,8.999999E+09,8.999999E+09]];
	LOCAL CONST Robtarget Tr_meulage_bavure_P208 :=[[-245.640640625,-63.9730234375,20],[0.523185325377564,-0.56182210386001,0.468956838300669,-0.436706449156553],[0,0,0,0],[8.999999E+09,8.999999E+09,8.999999E+09,8.999999E+09,8.999999E+09,8.999999E+09]];
	LOCAL CONST Robtarget Tr_meulage_bavure_P209 :=[[-245.49678125,-64.69972265625,20],[0.52430818698614,-0.562312145633216,0.467693041725851,-0.436083930744869],[0,0,0,0],[8.999999E+09,8.999999E+09,8.999999E+09,8.999999E+09,8.999999E+09,8.999999E+09]];
	LOCAL CONST Robtarget Tr_meulage_bavure_P210 :=[[-244.876265625,-70.7155,20],[0.525649903167548,-0.563074818500644,0.466134294580017,-0.435152556567009],[0,0,0,0],[8.999999E+09,8.999999E+09,8.999999E+09,8.999999E+09,8.999999E+09,8.999999E+09]];
	LOCAL CONST Robtarget Tr_meulage_bavure_P211 :=[[-244.868515625,-70.7529296875,20],[0.52716877954135,-0.564055033916588,0.464333917750362,-0.433968903744081],[0,0,0,0],[8.999999E+09,8.999999E+09,8.999999E+09,8.999999E+09,8.999999E+09,8.999999E+09]];
	LOCAL CONST Robtarget Tr_meulage_bavure_P212 :=[[-244.858625,-70.800046875,20],[0.528782992942236,-0.565181653870893,0.46239069102953,-0.43261194314541],[0,0,0,0],[8.999999E+09,8.999999E+09,8.999999E+09,8.999999E+09,8.999999E+09,8.999999E+09]];
	LOCAL CONST Robtarget Tr_meulage_bavure_P213 :=[[-244.797171875,-71.2724765625,20],[0.530396884089185,-0.566338749498168,0.460431253150214,-0.431210653031507],[0,0,0,0],[8.999999E+09,8.999999E+09,8.999999E+09,8.999999E+09,8.999999E+09,8.999999E+09]];
	LOCAL CONST Robtarget Tr_meulage_bavure_P214 :=[[-243.375765625,-79.1180078125,20],[0.531893569335625,-0.567416265757172,0.458605179079183,-0.42989452424443],[0,0,0,0],[8.999999E+09,8.999999E+09,8.999999E+09,8.999999E+09,8.999999E+09,8.999999E+09]];
	LOCAL CONST Robtarget Tr_meulage_bavure_P215 :=[[-243.05328125,-81.04115625,20],[0.533150445075168,-0.568290621079148,0.457074554337694,-0.428811409230941],[0,0,0,0],[8.999999E+09,8.999999E+09,8.999999E+09,8.999999E+09,8.999999E+09,8.999999E+09]];
	LOCAL CONST Robtarget Tr_meulage_bavure_P216 :=[[-242.70465625,-82.3746640625,20],[0.534074469084717,-0.56883436592015,0.455974510209037,-0.428111167408335],[0,0,0,0],[8.999999E+09,8.999999E+09,8.999999E+09,8.999999E+09,8.999999E+09,8.999999E+09]];
	LOCAL CONST Robtarget Tr_meulage_bavure_P217 :=[[-241.97528125,-85.75528125,20],[0.534576581970414,-0.568971279730662,0.455421582767437,-0.427891040803712],[0,0,0,0],[8.999999E+09,8.999999E+09,8.999999E+09,8.999999E+09,8.999999E+09,8.999999E+09]];
	LOCAL CONST Robtarget Tr_meulage_bavure_P218 :=[[-241.615421875,-86.7023046875,20],[0.534612055673805,-0.568649378823048,0.455477875280995,-0.428214594592361],[0,0,0,0],[8.999999E+09,8.999999E+09,8.999999E+09,8.999999E+09,8.999999E+09,8.999999E+09]];
	LOCAL CONST Robtarget Tr_meulage_bavure_P219 :=[[-241.147140625,-89.4847734375,20],[0.534164707859694,-0.567867331648727,0.456158274740717,-0.429085524002961],[0,0,0,0],[8.999999E+09,8.999999E+09,8.999999E+09,8.999999E+09,8.999999E+09,8.999999E+09]];
	LOCAL CONST Robtarget Tr_meulage_bavure_P220 :=[[-241.03396875,-89.851578125,20],[0.533266636416338,-0.566655043826004,0.457415976312859,-0.430464145319339],[0,0,0,0],[8.999999E+09,8.999999E+09,8.999999E+09,8.999999E+09,8.999999E+09,8.999999E+09]];
	LOCAL CONST Robtarget Tr_meulage_bavure_P221 :=[[-240.97271875,-90.152359375,20],[0.53199512047222,-0.565089414223428,0.45914289984932,-0.432253332253585],[0,0,0,0],[8.999999E+09,8.999999E+09,8.999999E+09,8.999999E+09,8.999999E+09,8.999999E+09]];
	LOCAL CONST Robtarget Tr_meulage_bavure_P222 :=[[-240.076328125,-97.31,20],[0.530454274431957,-0.563281012531,0.461195089337637,-0.434317686987033],[0,0,0,0],[8.999999E+09,8.999999E+09,8.999999E+09,8.999999E+09,8.999999E+09,8.999999E+09]];
	LOCAL CONST Robtarget Tr_meulage_bavure_P223 :=[[-239.742578125,-99.365953125,20],[0.528761934415614,-0.561363572008945,0.463411838242337,-0.43649882578453],[0,0,0,0],[8.999999E+09,8.999999E+09,8.999999E+09,8.999999E+09,8.999999E+09,8.999999E+09]];
	LOCAL CONST Robtarget Tr_meulage_bavure_P224 :=[[-239.600765625,-100.0753203125,20],[0.527054332838392,-0.559457139757307,0.46562216565305,-0.43865412099217],[0,0,0,0],[8.999999E+09,8.999999E+09,8.999999E+09,8.999999E+09,8.999999E+09,8.999999E+09]];
	LOCAL CONST Robtarget Tr_meulage_bavure_P225 :=[[-238.336875,-105.76425,20],[0.525435275045438,-0.557690981631371,0.46769068021236,-0.440640407120662],[0,0,0,0],[8.999999E+09,8.999999E+09,8.999999E+09,8.999999E+09,8.999999E+09,8.999999E+09]];
	LOCAL CONST Robtarget Tr_meulage_bavure_P226 :=[[-238.021953125,-107.32565625,20],[0.523999843509751,-0.556153942309196,0.469504538931484,-0.442360084522136],[0,0,0,0],[8.999999E+09,8.999999E+09,8.999999E+09,8.999999E+09,8.999999E+09,8.999999E+09]];
	LOCAL CONST Robtarget Tr_meulage_bavure_P227 :=[[-237.46903125,-109.0245078125,20],[0.522811743410168,-0.554913134716486,0.470989668015462,-0.443743198814617],[0,0,0,0],[8.999999E+09,8.999999E+09,8.999999E+09,8.999999E+09,8.999999E+09,8.999999E+09]];
	LOCAL CONST Robtarget Tr_meulage_bavure_P228 :=[[-236.995265625,-111.5783828125,20],[0.521909997676728,-0.554008393914595,0.472103437976193,-0.444750489205248],[0,0,0,0],[8.999999E+09,8.999999E+09,8.999999E+09,8.999999E+09,8.999999E+09,8.999999E+09]];
	LOCAL CONST Robtarget Tr_meulage_bavure_P229 :=[[-236.7246875,-112.6121953125,20],[0.521299580254171,-0.553452629691279,0.472842620958046,-0.445372641863147],[0,0,0,0],[8.999999E+09,8.999999E+09,8.999999E+09,8.999999E+09,8.999999E+09,8.999999E+09]];
	LOCAL CONST Robtarget Tr_meulage_bavure_P230 :=[[-235.45284375,-121.61003125,20],[0.520978748277058,-0.553230703704067,0.473215222344747,-0.445627967775794],[0,0,0,0],[8.999999E+09,8.999999E+09,8.999999E+09,8.999999E+09,8.999999E+09,8.999999E+09]];
	LOCAL CONST Robtarget Tr_meulage_bavure_P231 :=[[-235.4365625,-121.711515625,20],[0.520923193925815,-0.553320932498526,0.473251705667733,-0.445542135798255],[0,0,0,0],[8.999999E+09,8.999999E+09,8.999999E+09,8.999999E+09,8.999999E+09,8.999999E+09]];
	LOCAL CONST Robtarget Tr_meulage_bavure_P232 :=[[-235.392625,-122.0954921875,20],[0.521117283814843,-0.553680191235836,0.472977004205009,-0.445160393381693],[0,0,0,0],[8.999999E+09,8.999999E+09,8.999999E+09,8.999999E+09,8.999999E+09,8.999999E+09]];
	LOCAL CONST Robtarget Tr_meulage_bavure_P233 :=[[-234.22059375,-128.8344140625,20],[0.521503288264718,-0.554280282895751,0.472454368247833,-0.444516094473118],[0,0,0,0],[8.999999E+09,8.999999E+09,8.999999E+09,8.999999E+09,8.999999E+09,8.999999E+09]];
	LOCAL CONST Robtarget Tr_meulage_bavure_P234 :=[[-233.818265625,-131.326671875,20],[0.5220500190735,-0.555067966144619,0.471725290641918,-0.443664941948575],[0,0,0,0],[8.999999E+09,8.999999E+09,8.999999E+09,8.999999E+09,8.999999E+09,8.999999E+09]];
	LOCAL CONST Robtarget Tr_meulage_bavure_P235 :=[[-233.523953125,-133.01884375,20],[0.522714893701434,-0.555992134957476,0.470842445395975,-0.442661583358737],[0,0,0,0],[8.999999E+09,8.999999E+09,8.999999E+09,8.999999E+09,8.999999E+09,8.999999E+09]];
	LOCAL CONST Robtarget Tr_meulage_bavure_P236 :=[[-233.215234375,-134.5228125,20],[0.523448747419659,-0.556993398290956,0.469867648738029,-0.441570102876631],[0,0,0,0],[8.999999E+09,8.999999E+09,8.999999E+09,8.999999E+09,8.999999E+09,8.999999E+09]];
	LOCAL CONST Robtarget Tr_meulage_bavure_P237 :=[[-232.851921875,-136.650125,20],[0.524195318915837,-0.558019819928482,0.468869124019331,-0.440448513148874],[0,0,0,0],[8.999999E+09,8.999999E+09,8.999999E+09,8.999999E+09,8.999999E+09,8.999999E+09]];
	LOCAL CONST Robtarget Tr_meulage_bavure_P238 :=[[-232.60815625,-137.715671875,20],[0.52489555055306,-0.559009848538509,0.467921301424386,-0.439365799670232],[0,0,0,0],[8.999999E+09,8.999999E+09,8.999999E+09,8.999999E+09,8.999999E+09,8.999999E+09]];
	LOCAL CONST Robtarget Tr_meulage_bavure_P239 :=[[-232.417375,-139.0939375,20],[0.525509945158262,-0.559898574852785,0.467080801947005,-0.438392983372365],[0,0,0,0],[8.999999E+09,8.999999E+09,8.999999E+09,8.999999E+09,8.999999E+09,8.999999E+09]];
	LOCAL CONST Robtarget Tr_meulage_bavure_P240 :=[[-231.780015625,-142.52665625,20],[0.525982420745966,-0.560647331154684,0.46641552861573,-0.437576984999729],[0,0,0,0],[8.999999E+09,8.999999E+09,8.999999E+09,8.999999E+09,8.999999E+09,8.999999E+09]];
	LOCAL CONST Robtarget Tr_meulage_bavure_P241 :=[[-231.36753125,-144.0370625,20],[0.526299571311548,-0.561210222489061,0.465952249342011,-0.436967217013107],[0,0,0,0],[8.999999E+09,8.999999E+09,8.999999E+09,8.999999E+09,8.999999E+09,8.999999E+09]];
	LOCAL CONST Robtarget Tr_meulage_bavure_P242 :=[[-230.877484375,-147.175375,20],[0.526435167572928,-0.56157636640684,0.465721890888862,-0.436578881054337],[0,0,0,0],[8.999999E+09,8.999999E+09,8.999999E+09,8.999999E+09,8.999999E+09,8.999999E+09]];
	LOCAL CONST Robtarget Tr_meulage_bavure_P243 :=[[-230.8725,-147.201421875,20],[0.526390858856777,-0.561730134702477,0.465727791564854,-0.436428165501822],[0,0,0,0],[8.999999E+09,8.999999E+09,8.999999E+09,8.999999E+09,8.999999E+09,8.999999E+09]];
	LOCAL CONST Robtarget Tr_meulage_bavure_P244 :=[[-230.823625,-147.513625,20],[0.526172322715589,-0.561689860899808,0.465959941143116,-0.436495727608347],[0,0,0,0],[8.999999E+09,8.999999E+09,8.999999E+09,8.999999E+09,8.999999E+09,8.999999E+09]];
	LOCAL CONST Robtarget Tr_meulage_bavure_P245 :=[[-229.736046875,-152.626703125,20],[0.52581123170215,-0.561470555377054,0.466382182103955,-0.436761976683415],[0,0,0,0],[8.999999E+09,8.999999E+09,8.999999E+09,8.999999E+09,8.999999E+09,8.999999E+09]];
	LOCAL CONST Robtarget Tr_meulage_bavure_P246 :=[[-229.299703125,-154.8508125,20],[0.525346724693692,-0.561108241824334,0.466945072896379,-0.437184925069713],[0,0,0,0],[8.999999E+09,8.999999E+09,8.999999E+09,8.999999E+09,8.999999E+09,8.999999E+09]];
	LOCAL CONST Robtarget Tr_meulage_bavure_P247 :=[[-228.77840625,-156.91525,20],[0.524817917119832,-0.560643715749193,0.467597942658644,-0.43771787932679],[0,0,0,0],[8.999999E+09,8.999999E+09,8.999999E+09,8.999999E+09,8.999999E+09,8.999999E+09]];
	LOCAL CONST Robtarget Tr_meulage_bavure_P248 :=[[-228.337578125,-159.03828125,20],[0.524253168568131,-0.560132511970143,0.468297596484806,-0.438300747668591],[0,0,0,0],[8.999999E+09,8.999999E+09,8.999999E+09,8.999999E+09,8.999999E+09,8.999999E+09]];
	LOCAL CONST Robtarget Tr_meulage_bavure_P249 :=[[-227.9853125,-160.117296875,20],[0.523713869120416,-0.559599418193556,0.468975390438537,-0.438901307370324],[0,0,0,0],[8.999999E+09,8.999999E+09,8.999999E+09,8.999999E+09,8.999999E+09,8.999999E+09]];
	LOCAL CONST Robtarget Tr_meulage_bavure_P250 :=[[-227.521234375,-162.7755,20],[0.523220829574292,-0.559084901825633,0.469600315593168,-0.439476483608632],[0,0,0,0],[8.999999E+09,8.999999E+09,8.999999E+09,8.999999E+09,8.999999E+09,8.999999E+09]];
	LOCAL CONST Robtarget Tr_meulage_bavure_P251 :=[[-227.291359375,-163.6646875,20],[0.522793296500426,-0.558609612203602,0.470148106639312,-0.440003668293151],[0,0,0,0],[8.999999E+09,8.999999E+09,8.999999E+09,8.999999E+09,8.999999E+09,8.999999E+09]];
	LOCAL CONST Robtarget Tr_meulage_bavure_P252 :=[[-226.867859375,-166.444859375,20],[0.522447651822771,-0.558175665722447,0.470601994139436,-0.440479443802049],[0,0,0,0],[8.999999E+09,8.999999E+09,8.999999E+09,8.999999E+09,8.999999E+09,8.999999E+09]];
	LOCAL CONST Robtarget Tr_meulage_bavure_P253 :=[[-226.801171875,-166.929015625,20],[0.522181142525718,-0.557784680600011,0.47096469186787,-0.440902895763094],[0,0,0,0],[8.999999E+09,8.999999E+09,8.999999E+09,8.999999E+09,8.999999E+09,8.999999E+09]];
	LOCAL CONST Robtarget Tr_meulage_bavure_P254 :=[[-226.157421875,-171.8009375,20],[0.521994445569203,-0.557417703431872,0.471240251193611,-0.441293471910271],[0,0,0,0],[8.999999E+09,8.999999E+09,8.999999E+09,8.999999E+09,8.999999E+09,8.999999E+09]];
	LOCAL CONST Robtarget Tr_meulage_bavure_P255 :=[[-225.505765625,-175.540625,20],[0.521863540440543,-0.55708095082489,0.471451682945062,-0.44164756314868],[0,0,0,0],[8.999999E+09,8.999999E+09,8.999999E+09,8.999999E+09,8.999999E+09,8.999999E+09]];
	LOCAL CONST Robtarget Tr_meulage_bavure_P256 :=[[-225.471234375,-175.850984375,20],[0.521794971690925,-0.556770159549994,0.471593513657211,-0.441968952336233],[0,0,0,0],[8.999999E+09,8.999999E+09,8.999999E+09,8.999999E+09,8.999999E+09,8.999999E+09]];
	LOCAL CONST Robtarget Tr_meulage_bavure_P257 :=[[-225.3011875,-176.710015625,20],[0.521799751880624,-0.556496176896298,0.471652217634316,-0.442245644000882],[0,0,0,0],[8.999999E+09,8.999999E+09,8.999999E+09,8.999999E+09,8.999999E+09,8.999999E+09]];
	LOCAL CONST Robtarget Tr_meulage_bavure_P258 :=[[-224.726671875,-179.28975,20],[0.521911944814894,-0.556287652147039,0.471586874968133,-0.442445238742671],[0,0,0,0],[8.999999E+09,8.999999E+09,8.999999E+09,8.999999E+09,8.999999E+09,8.999999E+09]];
	LOCAL CONST Robtarget Tr_meulage_bavure_P259 :=[[-224.46675,-180.686859375,20],[0.522186443488294,-0.556190725748661,0.471331499548757,-0.442515324436731],[0,0,0,0],[8.999999E+09,8.999999E+09,8.999999E+09,8.999999E+09,8.999999E+09,8.999999E+09]];
	LOCAL CONST Robtarget Tr_meulage_bavure_P260 :=[[-223.64975,-183.24321875,20],[0.522669558059158,-0.556269672369746,0.470824471982563,-0.442385466829823],[0,0,0,0],[8.999999E+09,8.999999E+09,8.999999E+09,8.999999E+09,8.999999E+09,8.999999E+09]];
	LOCAL CONST Robtarget Tr_meulage_bavure_P261 :=[[-223.43253125,-185.064515625,20],[0.523408438970911,-0.556582038312709,0.47000430547102,-0.441990942758343],[0,0,0,0],[8.999999E+09,8.999999E+09,8.999999E+09,8.999999E+09,8.999999E+09,8.999999E+09]];
	LOCAL CONST Robtarget Tr_meulage_bavure_P262 :=[[-223.243,-185.780859375,20],[0.524449248315149,-0.557160027744365,0.468815276151776,-0.441291203483944],[0,0,0,0],[8.999999E+09,8.999999E+09,8.999999E+09,8.999999E+09,8.999999E+09,8.999999E+09]];
	LOCAL CONST Robtarget Tr_meulage_bavure_P263 :=[[-222.899125,-188.462765625,20],[0.525794358925822,-0.558016058041477,0.467249225597239,-0.440268704620729],[0,0,0,0],[8.999999E+09,8.999999E+09,8.999999E+09,8.999999E+09,8.999999E+09,8.999999E+09]];
	LOCAL CONST Robtarget Tr_meulage_bavure_P264 :=[[-222.791890625,-188.96646875,20],[0.527406553492306,-0.559115411411257,0.465348191044884,-0.438957110828657],[0,0,0,0],[8.999999E+09,8.999999E+09,8.999999E+09,8.999999E+09,8.999999E+09,8.999999E+09]];
	LOCAL CONST Robtarget Tr_meulage_bavure_P265 :=[[-221.86121875,-195.59528125,20],[0.529224125373564,-0.560373194514731,0.463191350662076,-0.437444260064964],[0,0,0,0],[8.999999E+09,8.999999E+09,8.999999E+09,8.999999E+09,8.999999E+09,8.999999E+09]];
	LOCAL CONST Robtarget Tr_meulage_bavure_P266 :=[[-221.43671875,-197.810796875,20],[0.531141059217696,-0.56168216105965,0.460910309285864,-0.435848611279736],[0,0,0,0],[8.999999E+09,8.999999E+09,8.999999E+09,8.999999E+09,8.999999E+09,8.999999E+09]];
	LOCAL CONST Robtarget Tr_meulage_bavure_P267 :=[[-221.224203125,-198.865734375,20],[0.533020422432929,-0.56291882018825,0.458675468265913,-0.434313764412707],[0,0,0,0],[8.999999E+09,8.999999E+09,8.999999E+09,8.999999E+09,8.999999E+09,8.999999E+09]];
	LOCAL CONST Robtarget Tr_meulage_bavure_P268 :=[[-220.474703125,-201.547796875,20],[0.53473910952756,-0.563944797459528,0.456650768914386,-0.433001645966738],[0,0,0,0],[8.999999E+09,8.999999E+09,8.999999E+09,8.999999E+09,8.999999E+09,8.999999E+09]];
	LOCAL CONST Robtarget Tr_meulage_bavure_P269 :=[[-220.20240625,-203.242265625,20],[0.536190677944437,-0.564641055686131,0.45498095079006,-0.432055979633785],[0,0,0,0],[8.999999E+09,8.999999E+09,8.999999E+09,8.999999E+09,8.999999E+09,8.999999E+09]];
